// ---- POUs/CommonFB/MainFB/FB_CoupleAxis.TcPOU
(****************************************************************
NAME:			FB_CoupleAxis
DATA:			2017.2.16
VERSION:		1.0.0
DESCRIPTION:	FB_CoupleAxis
HISTORY:
				2017.2.16		NEW

***************************************************************)
FUNCTION_BLOCK FB_CoupleAxis
VAR_INPUT
	Execute:BOOL;
	Reset:BOOL;
END_VAR
VAR_OUTPUT
	FbID:DINT:=1001;
	State:DINT;
	Busy:BOOL;
	InGear:BOOL;
	Error:BOOL;
	ErrorID:DINT;
END_VAR
VAR_IN_OUT
END_VAR
VAR
	Bottom_MC_GearIn: MC_GearIn;
	Top_MC_GearIn: MC_GearIn;
	fb_ton: TON;
END_VAR

IF Execute THEN
Busy:=TRUE;
InGear:=FALSE;
fb_ton(PT:=t#0.1s);
CASE State OF
	0:	(*Check*)
		IF LeftTopLin.NcToPlc.CoupleState=3 OR LeftBottomLin.NcToPlc.CoupleState=3 THEN	
			ErrorID:=1;
			State:=-100;
		ELSIF LeftTopLin.NcToPlc.CoupleState=2 OR LeftBottomLin.NcToPlc.CoupleState=2
			OR RightTopLin.NcToPlc.CoupleState=2 OR RightBottomLin.NcToPlc.CoupleState=2 THEN
			ErrorID:=2;
			State:=-100;
		ELSIF LeftTopLin.NcToPlc.CoupleState=1 AND LeftBottomLin.NcToPlc.CoupleState=1
			AND RightTopLin.NcToPlc.CoupleState=3 AND RightBottomLin.NcToPlc.CoupleState=3 THEN	
			ErrorID:=3;
			State:=-100;
		ELSIF LeftTopLin.Status.Moving OR  RightTopLin.Status.Moving OR LeftBottomLin.Status.Moving OR RightBottomLin.Status.Moving THEN	(*ÓÐÖáÔË¶¯*)
			ErrorID:=4;
			State:=-100;
		ELSIF  Top_MC_GearIn.Error OR Bottom_MC_GearIn.Error THEN		(*FB Error*)
			ErrorID:=5;
			State:=99;
		ELSIF Top_MC_GearIn.InGear OR Bottom_MC_GearIn.InGear THEN
			ErrorID:=6;
			State:=99;
		ELSIF LeftTopLin.NcToPlc.CoupleState=0 AND LeftBottomLin.NcToPlc.CoupleState=0
			AND RightTopLin.NcToPlc.CoupleState=0 AND RightBottomLin.NcToPlc.CoupleState=0 THEN
			State:=1;
		ELSE
			ErrorID:=7;
			State:=-100;
		END_IF
	1:	(*Couple*)
		IF LeftTopLin.NcToPlc.CoupleState=0 AND LeftBottomLin.NcToPlc.CoupleState=0
			AND RightTopLin.NcToPlc.CoupleState=0 AND RightBottomLin.NcToPlc.CoupleState=0 THEN	
			Top_MC_GearIn.Execute:=TRUE;
			Bottom_MC_GearIn.Execute:=TRUE;
			A_CoupleMC();
			fb_ton.IN:=TRUE;
			State:=2;
		ELSE
			ErrorID:=7;
			State:=99;
		END_IF
	2:	(*Couple Wait*)
		A_CoupleMC();
		IF NOT Top_MC_GearIn.InGear OR NOT Bottom_MC_GearIn.InGear THEN	
			IF NOT fb_ton.Q THEN
				State:=2;
			ELSE
				ErrorID:=8;
				State:=99;
			END_IF
		ELSIF  LeftTopLin.NcToPlc.CoupleState<>1 OR  RightTopLin.NcToPlc.CoupleState<>3
			OR LeftBottomLin.NcToPlc.CoupleState<>1 OR  RightBottomLin.NcToPlc.CoupleState<>3 THEN	
				ErrorID:=9;
				State:=-100;
		ELSIF   LeftTopLin.NcToPlc.CoupleState=1 AND  RightTopLin.NcToPlc.CoupleState=3
			AND LeftBottomLin.NcToPlc.CoupleState=1 AND  RightBottomLin.NcToPlc.CoupleState=3 THEN	
				State:=88;
		ELSE
				ErrorID:=10;
				State:=-100;
		END_IF
	88:	(*InGear*)
		Execute:=FALSE;
		State:=0;
		Busy:=FALSE;
		InGear:=TRUE;
		Error:=FALSE;
		ErrorID:=0;
		Bottom_MC_GearIn.Execute:=FALSE;
		Top_MC_GearIn.Execute:=FALSE;
		A_CoupleMC();
		fb_ton.IN:=FALSE;
	99:	(*FB Error*)
		Execute:=FALSE;
		State:=99;
		Busy:=FALSE;
		InGear:=FALSE;
		Error:=TRUE;
		Bottom_MC_GearIn.Execute:=FALSE;
		Top_MC_GearIn.Execute:=FALSE;
		A_CoupleMC();
		fb_ton.IN:=FALSE;
	-100:	(*Emergency Error*)
		FB_PlcEmergencyStop();
		Execute:=FALSE;
		State:=-100;
		Busy:=FALSE;
		InGear:=FALSE;
		Error:=TRUE;
		Bottom_MC_GearIn.Execute:=FALSE;
		Top_MC_GearIn.Execute:=FALSE;
		A_CoupleMC();
		fb_ton.IN:=FALSE;
END_CASE
END_IF
IF Reset THEN
		Execute:=FALSE;
		State:=0;
		Busy:=FALSE;
		InGear:=FALSE;
		Error:=FALSE;
		ErrorID:=0;
		Bottom_MC_GearIn.Execute:=FALSE;
		Top_MC_GearIn.Execute:=FALSE;
		A_CoupleMC();
		Reset:=FALSE;
END_IF

ACTION A_CoupleMC:
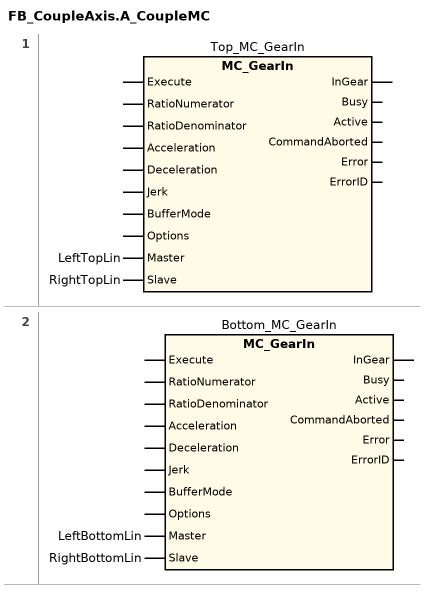
// NETWORK 1
Top_MC_GearIn(Master := LeftTopLin, Slave := RightTopLin); // MC_GearIn

// NETWORK 2
Bottom_MC_GearIn(Master := LeftBottomLin, Slave := RightBottomLin); // MC_GearIn
END_ACTION

END_FUNCTION_BLOCK

// ---- POUs/CommonFB/MainFB/FB_SetMotorAxisPosition.TcPOU
(****************************************************************
NAME:			FB_SetAxisPosition
DATA:			2017.2.16
VERSION:		1.0.0
DESCRIPTION:	FB_SetAxisPosition
HISTORY:
				2017.2.16		NEW

***************************************************************)
FUNCTION_BLOCK FB_SetMotorAxisPosition
VAR_INPUT
	//GapValueSet:LREAL:=0;
	ValueSet_LeftTop:LREAL:=0;
	ValueSet_RightTop:LREAL:=0;
	ValueSet_LeftBottom:LREAL:=0;
	ValueSet_RightBottom:LREAL:=0;
	Execute:BOOL;
END_VAR
VAR_OUTPUT
	FbID:DINT:=1001;
	State:DINT;
	Busy:BOOL;
	Done:BOOL;
	Error:BOOL;
	ErrorID:DINT;
END_VAR
VAR
	LeftTopMotor_MC_SetPosition: MC_SetPosition;
	RightTopMotor_MC_SetPosition: MC_SetPosition;
	LeftBottomMotor_MC_SetPosition: MC_SetPosition;
	RightBottomMotor_MC_SetPosition: MC_SetPosition;
	fb_ton: TON;
	FB_Couple_Axis: FB_CoupleAxis;
	FB_PlcEmergencyStop: FB_PlcEmergencyStop;
END_VAR

IF Execute THEN
Busy:=TRUE;
Done:=FALSE;
fb_ton(PT:=t#0.1s);
CASE State OF
	0:
		IF LeftTopMotor_MC_SetPosition.Error OR RightTopMotor_MC_SetPosition.Error
			OR LeftBottomMotor_MC_SetPosition.Error OR RightBottomMotor_MC_SetPosition.Error THEN		(*FB Error*)
			ErrorID:=1;
			State:=99;
		ELSIF FB_Couple_Axis.InGear THEN		
			ErrorID:=2;
			State:=99;
		ELSIF LeftTopMotor.NcToPlc.CoupleState=0 AND LeftBottomMotor.NcToPlc.CoupleState=0
			AND RightTopMotor.NcToPlc.CoupleState=0 AND RightBottomMotor.NcToPlc.CoupleState=0 THEN	
			State:=1;
		ELSE
			ErrorID:=3;
			State:=-100;
		END_IF
	1:	(*Execute*)
		LeftTopMotor_MC_SetPosition.Position:=ValueSet_LeftTop;
		LeftTopMotor_MC_SetPosition.Execute:=TRUE;
		RightTopMotor_MC_SetPosition.Position:=ValueSet_RightTop;
		RightTopMotor_MC_SetPosition.Execute:=TRUE;
		LeftBottomMotor_MC_SetPosition.Position:=ValueSet_LeftBottom;
		LeftBottomMotor_MC_SetPosition.Execute:=TRUE;
		RightBottomMotor_MC_SetPosition.Position:=ValueSet_RightBottom;
		RightBottomMotor_MC_SetPosition.Execute:=TRUE;
		A_SetMotorPositionMC();
		fb_ton.IN:=TRUE;
		State:=2;
	2:	(*Wait*)
		A_SetMotorPositionMC();
		IF NOT LeftTopMotor_MC_SetPosition.Done OR NOT RightTopMotor_MC_SetPosition.Done
			OR NOT LeftBottomMotor_MC_SetPosition.Done OR NOT RightBottomMotor_MC_SetPosition.Done THEN		
			IF NOT fb_ton.Q THEN
				State:=2;
			ELSE
				ErrorID:=4;
				State:=99;
			END_IF
		ELSIF  LeftTopMotor_MC_SetPosition.Done AND RightTopMotor_MC_SetPosition.Done
			AND LeftBottomMotor_MC_SetPosition.Done AND RightBottomMotor_MC_SetPosition.Done THEN		
			State:=88;
		ELSE
			ErrorID:=5;
			State:=99;
		END_IF
	88:
		Execute:=FALSE;
		State:=0;
		Busy:=FALSE;
		Done:=TRUE;
		Error:=FALSE;
		ErrorID:=0;
		LeftTopMotor_MC_SetPosition.Execute:=FALSE;
		RightTopMotor_MC_SetPosition.Execute:=FALSE;
		LeftBottomMotor_MC_SetPosition.Execute:=FALSE;
		RightBottomMotor_MC_SetPosition.Execute:=FALSE;
		fb_ton.IN:=FALSE;
	99:
		Execute:=FALSE;
		State:=99;
		Busy:=FALSE;
		Done:=FALSE;
		Error:=TRUE;
		LeftTopMotor_MC_SetPosition.Execute:=FALSE;
		RightTopMotor_MC_SetPosition.Execute:=FALSE;
		LeftBottomMotor_MC_SetPosition.Execute:=FALSE;
		RightBottomMotor_MC_SetPosition.Execute:=FALSE;
		fb_ton.IN:=FALSE;
	-100:
		FB_PlcEmergencyStop();
		Execute:=FALSE;
		State:=-100;
		Busy:=FALSE;
		Done:=FALSE;
		Error:=TRUE;
		LeftTopMotor_MC_SetPosition.Execute:=FALSE;
		RightTopMotor_MC_SetPosition.Execute:=FALSE;
		LeftBottomMotor_MC_SetPosition.Execute:=FALSE;
		RightBottomMotor_MC_SetPosition.Execute:=FALSE;
		fb_ton.IN:=FALSE;
END_CASE
END_IF

ACTION A_SetMotorPositionMC:
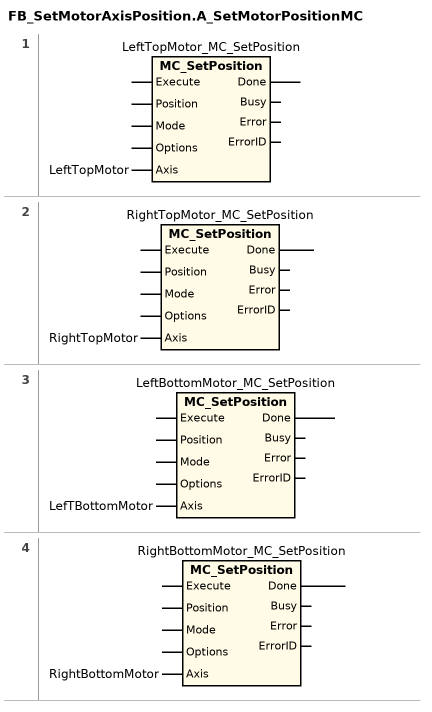
// NETWORK 1
LeftTopMotor_MC_SetPosition(Axis := LeftTopMotor); // MC_SetPosition

// NETWORK 2
RightTopMotor_MC_SetPosition(Axis := RightTopMotor); // MC_SetPosition

// NETWORK 3
LeftBottomMotor_MC_SetPosition(Axis := LefTBottomMotor); // MC_SetPosition

// NETWORK 4
RightBottomMotor_MC_SetPosition(Axis := RightBottomMotor); // MC_SetPosition
END_ACTION

END_FUNCTION_BLOCK

// ---- POUs/1.CarrierMode/SingleCarrierMode/SingleCarrierMode.TcPOU
PROGRAM SingleCarrierMode
VAR
	TopPositionNew:LREAL:=100;
	TopVelocityNew:LREAL:=0.02;
	btn_TopMove:BOOL;
	btn_TopStop:BOOL;
	BottomPositionNew:LREAL:=100;
	BottomVelocityNew:LREAL:=0.02;
	btn_BottomMove:BOOL;
	btn_BottomStop:BOOL;
	(*Var*)
	fb_ton1:TON;
	fb_ton2:TON;
	fb_ton3:TON;
	(*Status*)
	State:DINT;
	Busy:BOOL;
	TopBusy:BOOL;
	BottomBusy:BOOL;
	InitDone:BOOL;
	tm_state: DINT;
	ts_state: DINT;
	bm_state: DINT;
	bs_state: DINT;
	moni_State:DINT;
	(*PowerOff*)
	d_state: DINT;
	(*¼ì²âµ½ÏÞÎ»£¬»Ö¸´Move×´Ì¬*)
	FTrig_ReachLS: F_TRIG;
	FTrig_btn_GapMove: F_TRIG;
	InitPowerDone:BOOL;
END_VAR

TopPositionActual:=(Pos_LeftTopLin+Pos_RightTopLin)/2;
TopVelocityActual:=(Velo_LeftTopLin+Velo_RightTopLin)/2;
BottomPositionActual:=(Pos_LeftBottomLin+Pos_RightBOttomLin)/2;
BottomVelocityActual:=(Velo_LeftBottomLin+Velo_RightBOttomLin)/2;
(*btn_Power On/Off*)
IF btn_Power AND st_Power=0 THEN
	btn_PowerOn:=TRUE;
	btn_Power:=FALSE;
END_IF
IF btn_Power AND st_Power=1 THEN
	btn_PowerOff:=TRUE;
	btn_Power:=FALSE;
END_IF
IF btn_PowerOn THEN
	A_PowerOn();
END_IF
IF btn_PowerOff THEN
	A_PowerOff();
END_IF

(*********************************************************************Monitor All Carrirt Position***********************************************)
A_MonitoringAllAxis();
(*********************************************************************btn_TopMove*****************************************************************)
IF btn_TopMove AND NOT bottomBusy THEN
		TopBusy:=TRUE;
		btn_BottomMove:=FALSE;
		IF NOT st_Power THEN
			ErrorID:=1501;
			Error:=TRUE;
			ErrorDescription:='Plz PowerOn Frist';
			LED_Error:=TRUE;
			RETURN;
		ELSE
			ErrorID:=0;
			Error:=FALSE;
			ErrorDescription:='';
			LED_Error:=FALSE;
		END_IF
		CASE tm_state OF
			0:
				FB_Move.Mode:=2;						(*单梁模式*)
				FB_Move.CoupleState:=st_Couple;			
				FB_Move.PowerState:=st_Power;			
				FB_Move.TopMove:=TRUE;				
				FB_Move.TopPosition:=TopPositionNew;		
				FB_Move.TopVelocity:=TopVelocityNew;		
				FB_Move();								
				tm_state:=1;
			1:
				FB_Move();
				LED_Run:=TRUE;
				IF NOT FB_Move.TopDone THEN	
					tm_state:=1;
				ELSE					
					tm_state:=88;
				END_IF
			88:
				btn_TopMove:=FALSE;	
				LED_Run:=FALSE;
				tm_state:=0;
				TopBusy:=FALSE;
		END_CASE
END_IF

(*********************************************************************btn_BottomMove*****************************************************************)
IF btn_BottomMove AND NOT TopBusy THEN
		btn_TopMove:=FALSE;
		BottomBusy:=TRUE;
		IF NOT st_Power THEN
			ErrorID:=1501;
			Error:=TRUE;
			ErrorDescription:='Plz PowerOn Frist';
			LED_Error:=TRUE;
			RETURN;
		ELSE
			ErrorID:=0;
			Error:=FALSE;
			ErrorDescription:='';
			LED_Error:=FALSE;
		END_IF
		CASE bm_state OF
			0:
				FB_Move.Mode:=2;						
				FB_Move.CoupleState:=st_Couple;			
				FB_Move.PowerState:=st_Power;			
				FB_Move.BottomMove:=TRUE;			
				FB_Move.BottomPosition:=BottomPositionNew;		
				FB_Move.BottomVelocity:=BottomVelocityNew;		
				FB_Move();
				bm_state:=1;
			1:
				FB_Move();
				IF NOT FB_Move.BottomDone THEN
					LED_Run:=TRUE;
					bm_state:=1;
				ELSE
					bm_state:=88;
				END_IF
			88:
				BottomBusy:=FALSE;
				btn_TopMove:=FALSE;
				btn_BottomMove:=FALSE;
				bm_state:=0;
				LED_Run:=FALSE;
		END_CASE
END_IF
(*******************************************************************btn_TopStop********************************************************************)

IF btn_TopStop OR btn_reset THEN
	LED_Run:=FALSE;
	TopMoveIndicator:=0;
	FB_Move.TopReset:=TRUE;
	TopBusy:=FALSE;
	FB_Move();
	btn_TopMove:=FALSE;	
	tm_state:=0;
	CASE ts_state OF
			0:
				FB_Stop.Mode:=2;
				FB_Stop.CoupleState:=st_Couple;
				FB_Stop.PowerState:=st_Power;
				FB_Stop.TopStop:=TRUE;	
				FB_Stop();	
				ts_state:=1;
			1:
				FB_Stop();
				IF NOT FB_Stop.TopDone THEN
					ts_state:=1;
				ELSE
					ts_state:=88;
				END_IF
			88:
				btn_TopStop:=FALSE;	
				FB_Move.TopReset:=FALSE;	
				ts_state:=0;
				btn_reset:=FALSE;
		END_CASE
END_IF
(*******************************************************************btn_BottomStop********************************************************************)
IF btn_BottomStop OR btn_reset THEN
	LED_Run:=FALSE;
	BottomMoveIndicator:=0;
	FB_Move.BottomReset:=TRUE;
	BottomBusy:=FALSE;
	FB_Move();			
	btn_BottomMove:=FALSE;			
	bm_state:=0;							
	CASE bs_state OF
			0:
				FB_Stop.Mode:=2;							
				FB_Stop.CoupleState:=st_Couple;			
				FB_Stop.PowerState:=st_Power;			
				FB_Stop.BottomStop:=TRUE;				
				FB_Stop();								
				bs_state:=1;
			1:
				FB_Stop();
				IF NOT FB_Stop.BottomDone THEN		
					bs_state:=1;
				ELSE									
					bs_state:=88;
				END_IF
			88:
				btn_BottomStop:=FALSE;					
				FB_Move.BottomReset:=FALSE;				
				bs_state:=0;
				btn_reset:=FALSE;
		END_CASE
END_IF
(************************************************************************************************************************)

FTrig_ReachLS(CLK:=Unreach_LS_Far AND Unreach_LS_Near);
IF FTrig_ReachLS.Q THEN		
	btn_TopStop:=TRUE;
	btn_BottomStop:=TRUE;
END_IF
IF btn_TopStop THEN			
	btn_BottomStop:=TRUE;
END_IF

ACTION A_MonitoringAllAxis:
(****************************************************************
NAME:			A_MonitoringAllAxis
DATA:			2017.3.20
VERSION:		1.0.0
DESCRIPTION:	

HISTORY:
				2017.3.20		NEW

***************************************************************)
IF  st_Power<>0 THEN
		Diff_TopPos_actual:=Pos_leftTopLin-Pos_RightTopLin;
		Diff_TopVelo_actual:=Velo_leftTopLin-Velo_RightTopLin;
IF ABS(Pos_leftTopLin-Pos_RightTopLin)>Threshold_TopPos_SingleCarrier THEN
		btn_TopStop:=TRUE;
		btn_BottomStop:=TRUE;
		FB_PlcEmergencyStop();
		Error:=TRUE;
		ErrorID:=14;
		LED_Error:=TRUE;
ELSIF ABS(Velo_leftTopLin-Velo_RightTopLin)>Threshold_TopVelo_SingleCarrier  THEN
		(*btn_TopStop:=TRUE;
		btn_BottomStop:=TRUE;
		FB_PlcEmergencyStop();*)
		Error:=TRUE;
		ErrorID:=15;

ELSIF ABS(Pos_LeftBottomLin-Pos_RightBottomLin)>Threshold_BottomPos_SingleCarrier THEN
		btn_TopStop:=TRUE;
		btn_BottomStop:=TRUE;
		FB_PlcEmergencyStop();
		Error:=TRUE;
		ErrorID:=16;
		LED_Error:=TRUE;
ELSIF ABS(Velo_leftBottomLin-Velo_RightBottomLin)>Threshold_BottomVelo_SingleCarrier  THEN
		(*btn_TopStop:=TRUE;
		btn_BottomStop:=TRUE;
		FB_PlcEmergencyStop();*)
		Error:=TRUE;
		ErrorID:=17;

END_IF
END_IF
(**************************************************************************************************************************************)
END_ACTION

ACTION A_PowerOff:
CASE d_state OF
		0:(*PowerOff*)
			FB_Power(Off:=TRUE);
				d_state:=1;
		1:
			IF NOT FB_power.OffStatus THEN
				d_state:=1;
			ELSE
				d_state:=88;
			END_IF
		88:(*ResetAllState*)
			btn_PowerOn:=FALSE;
			btn_TopMove:=FALSE;
			btn_TopStop:=FALSE;
			btn_BottomMove:=FALSE;
			btn_BottomStop:=FALSE;
			LeftTopLinMoveIndicator:=0;
			RightTopLinMoveIndicator:=0;
			LeftBottomLinMoveIndicator:=0;
			RightBottomLinMoveIndicator:=0;
			fb_ton1.IN:=FALSE;
			fb_ton2.IN:=FALSE;
			fb_ton3.IN:=FALSE;
			State:=0;
			Busy:=FALSE;
			InitPowerDone:=FALSE;
			Error:=FALSE;
			ErrorID:=0;
			tm_state:=0;
			ts_state:=0;
			bm_state:=0;
			bs_state:=0;
			btn_PowerOff:=FALSE;
			d_state:=0;
			Led_Run:=FALSE;
			Led_Error:=FALSE;
			moni_State:=0;
END_CASE
END_ACTION

ACTION A_PowerOn:
(****************************************************************
NAME:			A_PowerOn
DATA:			2018.1.9
VERSION:		1.0.0
DESCRIPTION:	

HISTORY:
				2019.1.9		NEW

***************************************************************)
fb_ton3(PT:=t#0.5s);
CASE State OF
	0:	(*FB_Power_On*)
		FB_Power(On:=TRUE);
		fb_ton3.IN:=TRUE;
		State:=1;
	1:	(*wait*)
		FB_power();
		IF NOT FB_power.OnStatus THEN
			IF NOT fb_ton3.Q THEN
				State:=1;
			ELSE
				ErrorID:=1;
				State:=99;
			END_IF
		ELSE
			State:=88;
		END_IF
	88:	(*All Done*)
		btn_PowerOn:=FALSE;
		State:=0;
		Error:=FALSE;
		ErrorID:=0;
		Busy:=FALSE;
		InitPowerDone:=TRUE;
		FB_power.On:=FALSE;
		fb_ton3.IN:=FALSE;
		LED_Error:=FALSE;
	99:
		Error:=TRUE;
		//ErrorID:=701;
		//ErrorDescription:='power on error';		
		btn_PowerOn:=FALSE;
		State:=99;
		Busy:=FALSE;
		InitPowerDone:=FALSE;
		fb_ton3.IN:=FALSE;
		LED_Error:=TRUE;
END_CASE
END_ACTION

END_PROGRAM

// ---- POUs/CommonFB/MainFB/FB_Move.TcPOU
(****************************************************************
NAME:			FB_Move
DATA:			2017.2.17
VERSION:		1.0.0
DESCRIPTION:	FB_Move
HISTORY:
				2017.2.17		NEW
				2018.1.9		ÐÂÔöBCGapMode
***************************************************************)
FUNCTION_BLOCK FB_Move
VAR_INPUT
	(*È«¾Ö*)
	Mode:DINT;
	PowerState:BOOL;
	CoupleState:DINT;
	(*BCGapMode*)
	BCLeftTopPosition:LREAL;
	BCLeftTopVelocity:LREAL;
	BCRightTopPosition:LREAL;
	BCRightTopVelocity:LREAL;
	BCLeftBottomPosition:LREAL;
	BCLeftBottomVelocity:LREAL;
	BCRightBottomPosition:LREAL;
	BCRightBottomVelocity:LREAL;
	BCGapMove:BOOL;
	BCGapReset:BOOL;
	BCGapMove_2:BOOL;
	BCGapReset_2:BOOL;
	(*GapMode*)
	GapPosition:LREAL;
	GapVelocity:LREAL;
	GapMove:BOOL;
	GapReset:BOOL;
	(*SingleCarrierMode*)
	TopPosition:LREAL;
	TopVelocity:LREAL;
	TopMove:BOOL;
	TopReset:BOOL;
	BottomPosition:LREAL;
	BottomVelocity:LREAL;
	BottomMove:BOOL;
	BottomReset:BOOL;
	(*TaperMode*)
	TaperPosition:LREAL;
	TaperVelocity:LREAL;
	TaperMove:BOOL;
	TaperStop:BOOL;
	TaperReset:BOOL;
	(**DebugMode*)
	LeftTopPosition:LREAL;
	LeftTopVelocity:LREAL;
	LeftTopMove:BOOL;
	LeftTopStop:BOOL;
	LeftTopReset:BOOL;
	RightTopPosition:LREAL;
	RightTopVelocity:LREAL;
	RightTopMove:BOOL;
	RightTopStop:BOOL;
	RightTopReset:BOOL;
	LeftBottomPosition:LREAL;
	LeftBottomVelocity:LREAL;
	LeftBottomMove:BOOL;
	LeftBottomStop:BOOL;
	LeftBottomReset:BOOL;
	RightBottomPosition:LREAL;
	RightBottomVelocity:LREAL;
	RightBottomMove:BOOL;
	RightBottomStop:BOOL;
	RightBottomReset:BOOL;
END_VAR
VAR_OUTPUT
	FbID:DINT:=1001;
	GapState:DINT;
	GapBusy:BOOL;
	GapDone:BOOL;
	GapMoving:BOOL;

	BCGapState:DINT;
	BCGapBusy:BOOL;
	BCGapDone:BOOL;

	TopState:DINT;
	TopBusy:BOOL;
	TopDone:BOOL;
	BottomState:DINT;
	BottomBusy:BOOL;
	BottomDone:BOOL;

	TaperState:DINT;
	TaperBusy:BOOL;
	TaperDone:BOOL;

	LeftTopState:DINT;
	LeftTopBusy:BOOL;
	LeftTopDone:BOOL;
	RightTopState:DINT;
	RightTopBusy:BOOL;
	RightTopDone:BOOL;
	LeftBottomState:DINT;
	LeftBottomBusy:BOOL;
	LeftBottomDone:BOOL;
	RightBottomState:DINT;
	RightBottomBusy:BOOL;
	RightBottomDone:BOOL;


	Error:BOOL;
	ErrorID:DINT;
	
	GapState_2:DINT;
	GapBusy_2:BOOL;
	GapDone_2:BOOL;

	BCGapState_2:DINT;
	BCGapBusy_2:BOOL;
	BCGapDone_2:BOOL;
END_VAR
VAR
	Top_MC_MoveAbsolute: MC_MoveAbsolute;
	Bottom_MC_MoveAbsolute: MC_MoveAbsolute;
	RightTopLin_MC_MoveAbsolute: MC_MoveAbsolute;
	RightBottomLin_MC_MoveAbsolute: MC_MoveAbsolute;
	fb_ton: TON;
	fb_ton1: TON;
	fb_ton2: TON;
	fb_ton_debug_1:TON;
	fb_ton_debug_2:TON;
	fb_ton_debug_3:TON;
	fb_ton_debug_4:TON;
	fb_ton_BC:TON;
	fb_ton_BC_2:TON;
END_VAR

IF PowerState=1 THEN
	IF Mode=1 AND CoupleState=1 THEN
		A_GapMove();
	ELSIF Mode=2 AND CoupleState=0 AND TopMove THEN
		A_TopMove();
	ELSIF Mode=2 AND CoupleState=0 AND BottomMove THEN
		A_BottomMove();
	ELSIF Mode=3 AND CoupleState=0 AND TaperMove THEN
		A_TaperMove();
	ELSIF Mode=4 AND CoupleState=0 AND LeftTopMove THEN
		A_LeftTopMove();
	ELSIF Mode=4 AND CoupleState=0 AND RightTopMove THEN
		A_RightTopMove();
	ELSIF Mode=4 AND CoupleState=0 AND LeftBottomMove THEN
		A_LeftBottomMove();
	ELSIF Mode=4 AND CoupleState=0 AND RightBottomMove THEN
		A_RightBottomMove();
	ELSIF Mode=5 AND CoupleState=0 AND BCGapMove THEN
		A_BCGapMove();
	ELSIF Mode=6 AND CoupleState=0 AND BCGapMove_2 THEN
		A_BCGapMove_2();
	END_IF
END_IF

ACTION A_BCGapMove:
IF BCGapMove THEN
BCGapBusy:=TRUE;
BCGapDone:=FALSE;
fb_ton_BC(PT:=T#80S);(*2mm/s max spees,120mm*)

IF LeftTopLin.NcToPlc.CoupleState<>0 OR LeftBottomLin.NcToPlc.CoupleState<>0
			OR RightTopLin.NcToPlc.CoupleState<>0 OR RightBottomLin.NcToPlc.CoupleState<>0 THEN
			ErrorID:=1;
			GapState:=-100;
END_IF
A_MoveMC();
IF  LeftTopLin.Status.Moving AND RightTopLin.Status.Moving
			 AND LeftBottomLin.Status.Moving AND RightBottomLin.Status.Moving THEN
	GapMoving:=TRUE;
ELSE
	GapMoving:=FALSE;
END_IF
CASE BCGapState OF
	0:
		IF LeftTopLin.Status.Moving OR RightTopLin.Status.Moving
			 OR LeftBottomLin.Status.Moving OR RightBottomLin.Status.Moving THEN	
			BCGapState:=88;
		//ELSIF Top_MC_MoveAbsolute.Error OR Bottom_MC_MoveAbsolute.Error OR
		//		RightTopLin_MC_MoveAbsolute.Error OR RightBottomLin_MC_MoveAbsolute.Error THEN	
		//	ErrorID:=2;
		//	BCGapState:=99;
		(*ELSIF ABS(Pos_LeftTopLin-GapPosition/2)<0.002 AND  ABS(Pos_LeftBottomLin-GapPosition)<0.002 THEN	
			GapState:=88;*)
		ELSIF leftTopLin.Status.NotMoving AND  leftBottomLin.Status.NotMoving
			 AND RightTopLin.Status.NotMoving AND RightBottomLin.Status.NotMoving THEN	
			BCGapState:=1;
		END_IF
	1:
		Top_MC_MoveAbsolute.Position:=BCLeftTopPosition;
		Top_MC_MoveAbsolute.Velocity:=BCLeftTopVelocity;
		Bottom_MC_MoveAbsolute.Position:=BCLeftBottomPosition;
		Bottom_MC_MoveAbsolute.Velocity:=BCLeftBottomVelocity;
		RightTopLin_MC_MoveAbsolute.Position:=BCRightTopPosition;
		RightTopLin_MC_MoveAbsolute.Velocity:=BCRightTopVelocity;
		RightBottomLin_MC_MoveAbsolute.Position:=BCRightBottomPosition;
		RightBottomLin_MC_MoveAbsolute.Velocity:=BCRightBottomVelocity;
		Top_MC_MoveAbsolute.Execute:=TRUE;
		Bottom_MC_MoveAbsolute.Execute:=TRUE;
		RightTopLin_MC_MoveAbsolute.Execute:=TRUE;
		RightBottomLin_MC_MoveAbsolute.Execute:=TRUE;
		fb_ton_BC.IN:=TRUE;
		BCGapState:=2;
	2:
		IF NOT Top_MC_MoveAbsolute.Done OR NOT  Bottom_MC_MoveAbsolute.Done
				OR NOT RightTopLin_MC_MoveAbsolute.Done OR NOT RightBottomLin_MC_MoveAbsolute.Done THEN	
			BCGapState:=2;
		ELSIF Top_MC_MoveAbsolute.Done  AND  Bottom_MC_MoveAbsolute.Done AND RightTopLin_MC_MoveAbsolute.Done AND RightBottomLin_MC_MoveAbsolute.Done THEN		(*ÔË¶¯Íê³É£¬×ªÏÂÒ»²½*)
			BCGapState:=88;
		END_IF
		(*½ÓÊÕµ½stopÐÅºÅÊ±£¬reset×´Ì¬*)
		IF BCGapReset THEN
			BCGapState:=88;
		END_IF

	88:
		BCGapMove:=FALSE;
		BCGapState:=0;
		BCGapBusy:=FALSE;
		BCGapDone:=TRUE;
		Error:=FALSE;
		ErrorID:=0;
		Top_MC_MoveAbsolute.Execute:=FALSE;
		Bottom_MC_MoveAbsolute.Execute:=FALSE;
		RightTopLin_MC_MoveAbsolute.Execute:=FALSE;
		RightBottomLin_MC_MoveAbsolute.Execute:=FALSE;
		fb_ton_BC.IN:=FALSE;
	89:
		BCGapMove:=FALSE;
		BCGapState:=0;
		BCGapBusy:=FALSE;
		BCGapDone:=FALSE;
		Error:=FALSE;
		ErrorID:=0;
		Top_MC_MoveAbsolute.Execute:=FALSE;
		Bottom_MC_MoveAbsolute.Execute:=FALSE;
		RightTopLin_MC_MoveAbsolute.Execute:=FALSE;
		RightBottomLin_MC_MoveAbsolute.Execute:=FALSE;
		fb_ton_BC.IN:=FALSE;
	99:
		BCGapMove:=FALSE;
		BCGapState:=0;
		BCGapBusy:=FALSE;
		BCGapDone:=FALSE;
		Error:=TRUE;
		Top_MC_MoveAbsolute.Execute:=FALSE;
		Bottom_MC_MoveAbsolute.Execute:=FALSE;
		RightTopLin_MC_MoveAbsolute.Execute:=FALSE;
		RightBottomLin_MC_MoveAbsolute.Execute:=FALSE;
		fb_ton_BC.IN:=FALSE;
	-100:
		FB_PlcEmergencyStop();
		BCGapMove:=FALSE;
		BCGapState:=-100;
		BCGapBusy:=FALSE;
		BCGapDone:=FALSE;
		Error:=TRUE;
		Top_MC_MoveAbsolute.Execute:=FALSE;
		Bottom_MC_MoveAbsolute.Execute:=FALSE;
		RightTopLin_MC_MoveAbsolute.Execute:=FALSE;
		RightBottomLin_MC_MoveAbsolute.Execute:=FALSE;
		fb_ton_BC.IN:=FALSE;
END_CASE
END_IF
END_ACTION

ACTION A_BCGapMove_2:
IF BCGapMove_2 THEN
BCGapBusy_2:=TRUE;
BCGapDone_2:=FALSE;
fb_ton_BC_2(PT:=T#80S);(*2mm/s max spees,120mm*)
IF LeftTopLin.NcToPlc.CoupleState<>0 OR LeftBottomLin.NcToPlc.CoupleState<>0
			OR RightTopLin.NcToPlc.CoupleState<>0 OR RightBottomLin.NcToPlc.CoupleState<>0 THEN
			ErrorID:=1;
			GapState:=-100;
END_IF
A_MoveMC();
CASE BCGapState_2 OF
	0:
		IF LeftTopLin.Status.Moving OR RightTopLin.Status.Moving
			 OR LeftBottomLin.Status.Moving OR RightBottomLin.Status.Moving THEN	
			BCGapState_2:=88;
		ELSIF Top_MC_MoveAbsolute.Error OR Bottom_MC_MoveAbsolute.Error OR
				RightTopLin_MC_MoveAbsolute.Error OR RightBottomLin_MC_MoveAbsolute.Error THEN	
			ErrorID:=2;
			BCGapState_2:=99;
		(*ELSIF ABS(Pos_LeftTopLin-GapPosition/2)<0.002 AND  ABS(Pos_LeftBottomLin-GapPosition)<0.002 THEN	
			GapState:=88;*)
		ELSIF leftTopLin.Status.NotMoving AND  leftBottomLin.Status.NotMoving
			 AND RightTopLin.Status.NotMoving AND RightBottomLin.Status.NotMoving THEN
			BCGapState_2:=1;
		END_IF
	1:
		Top_MC_MoveAbsolute.Position:=BCLeftTopPosition;
		Top_MC_MoveAbsolute.Velocity:=BCLeftTopVelocity;
		Bottom_MC_MoveAbsolute.Position:=BCLeftBottomPosition;
		Bottom_MC_MoveAbsolute.Velocity:=BCLeftBottomVelocity;
		RightTopLin_MC_MoveAbsolute.Position:=BCRightTopPosition;
		RightTopLin_MC_MoveAbsolute.Velocity:=BCRightTopVelocity;
		RightBottomLin_MC_MoveAbsolute.Position:=BCRightBottomPosition;
		RightBottomLin_MC_MoveAbsolute.Velocity:=BCRightBottomVelocity;
		Top_MC_MoveAbsolute.Execute:=TRUE;
		Bottom_MC_MoveAbsolute.Execute:=TRUE;
		RightTopLin_MC_MoveAbsolute.Execute:=TRUE;
		RightBottomLin_MC_MoveAbsolute.Execute:=TRUE;
		fb_ton_BC_2.IN:=TRUE;
		BCGapState_2:=2;
	2:
		IF NOT Top_MC_MoveAbsolute.Done OR NOT  Bottom_MC_MoveAbsolute.Done
				OR NOT RightTopLin_MC_MoveAbsolute.Done OR NOT RightBottomLin_MC_MoveAbsolute.Done THEN		
			BCGapState_2:=2;
		ELSIF Top_MC_MoveAbsolute.Done  AND  Bottom_MC_MoveAbsolute.Done AND RightTopLin_MC_MoveAbsolute.Done AND RightBottomLin_MC_MoveAbsolute.Done THEN		(*ÔË¶¯Íê³É£¬×ªÏÂÒ»²½*)
			BCGapState_2:=88;
		END_IF
		(*½ÓÊÕµ½stopÐÅºÅÊ±£¬reset×´Ì¬*)
		IF BCGapReset_2 THEN
			BCGapState_2:=89;
		END_IF

	88:
		BCGapMove_2:=FALSE;
		BCGapState_2:=0;
		BCGapBusy_2:=FALSE;
		BCGapDone_2:=TRUE;
		Error:=FALSE;
		ErrorID:=0;
		Top_MC_MoveAbsolute.Execute:=FALSE;
		Bottom_MC_MoveAbsolute.Execute:=FALSE;
		RightTopLin_MC_MoveAbsolute.Execute:=FALSE;
		RightBottomLin_MC_MoveAbsolute.Execute:=FALSE;
		fb_ton_BC_2.IN:=FALSE;
	89:
		BCGapMove_2:=FALSE;
		BCGapState_2:=0;
		BCGapBusy_2:=FALSE;
		BCGapDone_2:=FALSE;
		Error:=FALSE;
		ErrorID:=0;
		Top_MC_MoveAbsolute.Execute:=FALSE;
		Bottom_MC_MoveAbsolute.Execute:=FALSE;
		RightTopLin_MC_MoveAbsolute.Execute:=FALSE;
		RightBottomLin_MC_MoveAbsolute.Execute:=FALSE;
		fb_ton_BC_2.IN:=FALSE;
	99:
		BCGapMove_2:=FALSE;
		BCGapState_2:=99;
		BCGapBusy_2:=FALSE;
		BCGapDone_2:=FALSE;
		Error:=TRUE;
		Top_MC_MoveAbsolute.Execute:=FALSE;
		Bottom_MC_MoveAbsolute.Execute:=FALSE;
		RightTopLin_MC_MoveAbsolute.Execute:=FALSE;
		RightBottomLin_MC_MoveAbsolute.Execute:=FALSE;
		fb_ton_BC_2.IN:=FALSE;
	-100:
		FB_PlcEmergencyStop();
		BCGapMove_2:=FALSE;
		BCGapState_2:=-100;
		BCGapBusy_2:=FALSE;
		BCGapDone_2:=FALSE;
		Error:=TRUE;
		Top_MC_MoveAbsolute.Execute:=FALSE;
		Bottom_MC_MoveAbsolute.Execute:=FALSE;
		RightTopLin_MC_MoveAbsolute.Execute:=FALSE;
		RightBottomLin_MC_MoveAbsolute.Execute:=FALSE;
		fb_ton_BC_2.IN:=FALSE;
END_CASE
END_IF
END_ACTION

ACTION A_BottomMove:
IF BottomMove THEN
BottomBusy:=TRUE;
BottomDone:=FALSE;
fb_ton2(PT:=T#80S);(*2mm/s max spees,120mm*)
A_MoveMC();
CASE BottomState OF

	0:
		IF LeftTopLin.Status.Moving OR RightTopLin.Status.Moving
			 OR LeftBottomLin.Status.Moving OR RightBottomLin.Status.Moving THEN	
			TopState:=88;
		ELSIF  Bottom_MC_MoveAbsolute.Error OR RightBottomLin_MC_MoveAbsolute.Error THEN		
			ErrorID:=2;
			BottomState:=99;
		ELSIF leftTopLin.Status.NotMoving AND  leftBottomLin.Status.NotMoving
			 AND RightTopLin.Status.NotMoving AND RightBottomLin.Status.NotMoving THEN	
			BottomState:=1;
		END_IF
	1:
		Bottom_MC_MoveAbsolute.Position:=BottomPosition;
		Bottom_MC_MoveAbsolute.Velocity:=BottomVelocity;
		Bottom_MC_MoveAbsolute.Execute:=TRUE;
		RightBottomLin_MC_MoveAbsolute.Position:=BottomPosition;
		RightBottomLin_MC_MoveAbsolute.Velocity:=BottomVelocity;
		RightBottomLin_MC_MoveAbsolute.Execute:=TRUE;
		fb_ton2.IN:=TRUE;
		BottomState:=2;
	2:
		IF leftTopLin.Status.Moving OR RightTopLin.Status.Moving THEN	
			ErrorID:=3;
			BottomState:=-100;
		ELSIF  (LeftBottomLin.Status.Moving AND  RightBottomLin.Status.NotMoving)
				OR (RightBottomLin.Status.Moving AND  LeftBottomLin.Status.NotMoving) THEN
			//ErrorID:=4;
			//BottomState:=-100;
		ELSIF NOT Bottom_MC_MoveAbsolute.Done THEN		
			BottomState:=2;
		ELSIF Bottom_MC_MoveAbsolute.Done THEN		
				BottomState:=88;
		END_IF
		(*½ÓÊÕµ½stopÐÅºÅÊ±£¬reset×´Ì¬*)
		IF BottomReset THEN
			BottomState:=89;
		END_IF

	88:
		BottomMove:=FALSE;
		BottomState:=0;
		BottomBusy:=FALSE;
		BottomDone:=TRUE;
		Error:=FALSE;
		ErrorID:=0;
		Bottom_MC_MoveAbsolute.Execute:=FALSE;
		RightBottomLin_MC_MoveAbsolute.Execute:=FALSE;
		fb_ton2.IN:=FALSE;
	89:
		BottomMove:=FALSE;
		BottomState:=0;
		BottomBusy:=FALSE;
		BottomDone:=FALSE;
		Error:=FALSE;
		ErrorID:=0;
		Bottom_MC_MoveAbsolute.Execute:=FALSE;
		RightBottomLin_MC_MoveAbsolute.Execute:=FALSE;
		fb_ton2.IN:=FALSE;
	99:
		BottomMove:=FALSE;
		BottomState:=99;
		BottomBusy:=FALSE;
		BottomDone:=FALSE;
		Error:=TRUE;
		Bottom_MC_MoveAbsolute.Execute:=FALSE;
		RightBottomLin_MC_MoveAbsolute.Execute:=FALSE;
		fb_ton2.IN:=FALSE;
	-100:
		FB_PlcEmergencyStop();
		BottomMove:=FALSE;
		BottomState:=-100;
		BottomBusy:=FALSE;
		BottomDone:=FALSE;
		Error:=TRUE;
		Bottom_MC_MoveAbsolute.Execute:=FALSE;
		RightBottomLin_MC_MoveAbsolute.Execute:=FALSE;
		fb_ton2.IN:=FALSE;
END_CASE
END_IF
END_ACTION

ACTION A_GapMove:
IF GapMove THEN
GapBusy:=TRUE;
GapDone:=FALSE;
fb_ton(PT:=T#80S);(*2mm/s max spees,120mm*)

IF LeftTopLin.NcToPlc.CoupleState<>1 OR LeftBottomLin.NcToPlc.CoupleState<>1
			OR RightTopLin.NcToPlc.CoupleState<>3 OR RightBottomLin.NcToPlc.CoupleState<>3 THEN
			ErrorID:=1;
			GapState:=-100;
END_IF
A_MoveMC();
CASE GapState OF

	0:
		IF LeftTopLin.Status.Moving OR RightTopLin.Status.Moving
			 OR LeftBottomLin.Status.Moving OR RightBottomLin.Status.Moving THEN	
			GapState:=88;
		ELSIF Top_MC_MoveAbsolute.Error OR Bottom_MC_MoveAbsolute.Error THEN		
			ErrorID:=2;
			GapState:=99;
		ELSIF ABS(Pos_LeftTopLin-GapPosition/2)<0.002 AND  ABS(Pos_LeftBottomLin-GapPosition)<0.002 THEN	
			GapState:=88;
		ELSIF leftTopLin.Status.NotMoving AND  leftBottomLin.Status.NotMoving
			 AND RightTopLin.Status.NotMoving AND RightBottomLin.Status.NotMoving THEN	
			GapState:=1;
		END_IF
	1:
		Top_MC_MoveAbsolute.Position:=GapPosition/2;
		Top_MC_MoveAbsolute.Velocity:=GapVelocity/2;
		Bottom_MC_MoveAbsolute.Position:=GapPosition/2;
		Bottom_MC_MoveAbsolute.Velocity:=GapVelocity/2;
		Top_MC_MoveAbsolute.Execute:=TRUE;
		Bottom_MC_MoveAbsolute.Execute:=TRUE;
		fb_ton.IN:=TRUE;
		GapState:=2;
	2:
		(*IF leftTopLin.Status.Moving AND   leftBottomLin.Status.NotMoving THEN (*ÉÏÏÂÁº²»Í¬Ê±¶¯*)
			ErrorID:=3;
			GapState:=-100;
		ELSIF RightTopLin.Status.NotMoving AND RightBottomLin.Status.Moving THEN (*ÉÏÏÂÁº²»Í¬Ê±¶¯*)
			ErrorID:=4;
			GapState:=-100;
		*)
		IF  (LeftTopLin.Status.Moving AND  RightTopLin.Status.NotMoving)
			OR  (LeftTopLin.Status.Moving AND LeftBottomLin.Status.NotMoving)
			OR (LeftTopLin.Status.Moving AND  RightBottomLin.Status.NotMoving)
				OR (RightTopLin.Status.Moving AND  LeftTopLin.Status.NotMoving)
				OR (RightTopLin.Status.Moving AND  LeftBottomLin.Status.NotMoving)
				OR (RightTopLin.Status.Moving AND  RightBottomLin.Status.NotMoving)
					OR (LeftBottomLin.Status.Moving AND  LeftTopLin.Status.NotMoving)
					OR (LeftBottomLin.Status.Moving AND  RightTopLin.Status.NotMoving)
					OR (LeftBottomLin.Status.Moving AND  RightBottomLin.Status.NotMoving)
						OR (RightBottomLin.Status.Moving AND  LeftTopLin.Status.NotMoving)
						OR (RightBottomLin.Status.Moving AND  RightTopLin.Status.NotMoving)
						OR (RightBottomLin.Status.Moving AND  LeftBottomLin.Status.NotMoving) THEN			
			ErrorID:=5;
			GapState:=-100;
		ELSIF NOT Top_MC_MoveAbsolute.Done OR NOT  Bottom_MC_MoveAbsolute.Done THEN		
			(*IF NOT  fb_ton.Q THEN
				GapState:=2;
			ELSE
				ErrorID:=5;
				GapState:=-100;
			END_IF*)
			GapState:=2;
		ELSIF Top_MC_MoveAbsolute.Done  AND  Bottom_MC_MoveAbsolute.Done THEN		
				GapState:=88;
		END_IF
		(*½ÓÊÕµ½stopÐÅºÅÊ±£¬reset×´Ì¬*)
		IF GapReset THEN
			GapState:=89;
		END_IF

	88:
		GapMove:=FALSE;
		GapState:=0;
		GapBusy:=FALSE;
		GapDone:=TRUE;
		Error:=FALSE;
		ErrorID:=0;
		Top_MC_MoveAbsolute.Execute:=FALSE;
		Bottom_MC_MoveAbsolute.Execute:=FALSE;
		fb_ton.IN:=FALSE;
	89:
		GapMove:=FALSE;
		GapState:=0;
		GapBusy:=FALSE;
		GapDone:=FALSE;
		Error:=FALSE;
		ErrorID:=0;
		Top_MC_MoveAbsolute.Execute:=FALSE;
		Bottom_MC_MoveAbsolute.Execute:=FALSE;
		fb_ton.IN:=FALSE;
	99:
		GapMove:=FALSE;
		GapState:=99;
		GapBusy:=FALSE;
		GapDone:=FALSE;
		Error:=TRUE;
		Top_MC_MoveAbsolute.Execute:=FALSE;
		Bottom_MC_MoveAbsolute.Execute:=FALSE;
		fb_ton.IN:=FALSE;
	-100:
		FB_PlcEmergencyStop();
		GapMove:=FALSE;
		GapState:=-100;
		GapBusy:=FALSE;
		GapDone:=FALSE;
		Error:=TRUE;
		Top_MC_MoveAbsolute.Execute:=FALSE;
		Bottom_MC_MoveAbsolute.Execute:=FALSE;
		fb_ton.IN:=FALSE;
END_CASE
END_IF
END_ACTION

ACTION A_LeftBottomMove:
IF LeftBottomMove THEN
LeftBottomBusy:=TRUE;
LeftBottomDone:=FALSE;
fb_ton_debug_3(PT:=t#10s);

IF LeftTopLin.NcToPlc.CoupleState<>0 OR LeftBottomLin.NcToPlc.CoupleState<>0
			OR RightTopLin.NcToPlc.CoupleState<>0 OR RightBottomLin.NcToPlc.CoupleState<>0 THEN
			ErrorID:=1;
			LeftBottomState:=-100;
END_IF
A_MoveMC();
CASE LeftBottomState OF
	0:
		IF Top_MC_MoveAbsolute.Error OR Bottom_MC_MoveAbsolute.Error
			OR RightTopLin_MC_MoveAbsolute.Error OR RightBottomLin_MC_MoveAbsolute.Error THEN	
			ErrorID:=2;
			LeftBottomState:=99;
		ELSIF leftTopLin.Status.NotMoving AND  leftBottomLin.Status.NotMoving
			 AND RightTopLin.Status.NotMoving AND RightBottomLin.Status.NotMoving THEN	
			LeftBottomState:=1;
		END_IF
	1:
		Bottom_MC_MoveAbsolute.Position:=LeftBottomPosition;
		Bottom_MC_MoveAbsolute.Velocity:=LeftBottomVelocity;
		Bottom_MC_MoveAbsolute.Execute:=TRUE;
		fb_ton_debug_3.IN:=TRUE;
		LeftBottomState:=2;
	2:
		IF LeftTopLin.Status.Moving OR RightTopLin.Status.Moving OR RightBottomLin.Status.Moving THEN	
			ErrorID:=3;
			LeftBottomState:=-100;
		ELSIF NOT Bottom_MC_MoveAbsolute.Done THEN		(*ÔË¶¯ÖÐ£¬¼ì²éDoneÐÅºÅ£¬Ã»ÓÐÔòÑ­»·£¬³¬Ê±±¨´í*)
			(*IF NOT  fb_ton.Q THEN
				LeftBottomState:=2;
			ELSE
				ErrorID:=5;
				LeftBottomState:=-100;
			END_IF*)
			LeftBottomState:=2;
		ELSIF Bottom_MC_MoveAbsolute.Done THEN		
				LeftBottomState:=88;
		END_IF

		IF LeftBottomReset THEN
			LeftBottomState:=89;
		END_IF

	88:
		LeftBottomMove:=FALSE;
		LeftBottomState:=0;
		LeftBottomBusy:=FALSE;
		LeftBottomDone:=TRUE;
		Error:=FALSE;
		ErrorID:=0;
		Bottom_MC_MoveAbsolute.Execute:=FALSE;
		fb_ton_debug_3.IN:=FALSE;
	89:
		LeftBottomMove:=FALSE;
		LeftBottomState:=0;
		LeftBottomBusy:=FALSE;
		LeftBottomDone:=FALSE;
		Error:=FALSE;
		ErrorID:=0;
		Bottom_MC_MoveAbsolute.Execute:=FALSE;
		fb_ton_debug_3.IN:=FALSE;
	99:
		LeftBottomMove:=FALSE;
		LeftBottomState:=99;
		LeftBottomBusy:=FALSE;
		LeftBottomDone:=FALSE;
		Error:=TRUE;
		Bottom_MC_MoveAbsolute.Execute:=FALSE;
		fb_ton_debug_3.IN:=FALSE;
	-100:
		FB_PlcEmergencyStop();
		LeftBottomMove:=FALSE;
		LeftBottomState:=-100;
		LeftBottomBusy:=FALSE;
		LeftBottomDone:=FALSE;
		Error:=TRUE;
		Bottom_MC_MoveAbsolute.Execute:=FALSE;
		fb_ton_debug_3.IN:=FALSE;
END_CASE
END_IF
END_ACTION

ACTION A_LeftTopMove:
IF LeftTopMove THEN
LeftTopBusy:=TRUE;
LeftTopDone:=FALSE;
fb_ton_debug_1(PT:=t#10s);

IF LeftTopLin.NcToPlc.CoupleState<>0 OR LeftBottomLin.NcToPlc.CoupleState<>0
			OR RightTopLin.NcToPlc.CoupleState<>0 OR RightBottomLin.NcToPlc.CoupleState<>0 THEN
			ErrorID:=1;
			LeftTopState:=-100;
END_IF
A_MoveMC();
CASE LeftTopState OF
	0:
		IF Top_MC_MoveAbsolute.Error OR Bottom_MC_MoveAbsolute.Error
			OR RightTopLin_MC_MoveAbsolute.Error OR RightBottomLin_MC_MoveAbsolute.Error THEN		
			ErrorID:=2;
			LeftTopState:=99;
		ELSIF leftTopLin.Status.NotMoving AND  leftBottomLin.Status.NotMoving
			 AND RightTopLin.Status.NotMoving AND RightBottomLin.Status.NotMoving THEN
			LeftTopState:=1;
		END_IF
	1:
		Top_MC_MoveAbsolute.Position:=LeftTopPosition;
		Top_MC_MoveAbsolute.Velocity:=LeftTopVelocity;
		Top_MC_MoveAbsolute.Execute:=TRUE;
		fb_ton_debug_1.IN:=TRUE;
		LeftTopState:=2;
	2:
		IF RightTopLin.Status.Moving OR LeftBottomLin.Status.Moving OR RightBottomLin.Status.Moving THEN
			ErrorID:=3;
			LeftTopState:=-100;
		ELSIF NOT Top_MC_MoveAbsolute.Done THEN	
			(*IF NOT  fb_ton.Q THEN
				LeftTopState:=2;
			ELSE
				ErrorID:=5;
				LeftTopState:=-100;
			END_IF*)
			LeftTopState:=2;
		ELSIF Top_MC_MoveAbsolute.Done THEN		
				LeftTopState:=88;
		END_IF
		(*½ÓÊÕµ½stopÐÅºÅÊ±£¬reset×´Ì¬*)
		IF LeftTopReset THEN
			LeftTopState:=89;
		END_IF

	88:
		LeftTopMove:=FALSE;
		LeftTopState:=0;
		LeftTopBusy:=FALSE;
		LeftTopDone:=TRUE;
		Error:=FALSE;
		ErrorID:=0;
		Top_MC_MoveAbsolute.Execute:=FALSE;
		fb_ton_debug_1.IN:=FALSE;
	89:
		LeftTopMove:=FALSE;
		LeftTopState:=0;
		LeftTopBusy:=FALSE;
		LeftTopDone:=FALSE;
		Error:=FALSE;
		ErrorID:=0;
		Top_MC_MoveAbsolute.Execute:=FALSE;
		fb_ton_debug_1.IN:=FALSE;
	99:
		LeftTopMove:=FALSE;
		LeftTopState:=99;
		LeftTopBusy:=FALSE;
		LeftTopDone:=FALSE;
		Error:=TRUE;
		Top_MC_MoveAbsolute.Execute:=FALSE;
		fb_ton_debug_1.IN:=FALSE;
	-100:
		FB_PlcEmergencyStop();
		LeftTopMove:=FALSE;
		LeftTopState:=-100;
		LeftTopBusy:=FALSE;
		LeftTopDone:=FALSE;
		Error:=TRUE;
		Top_MC_MoveAbsolute.Execute:=FALSE;
		fb_ton_debug_1.IN:=FALSE;
END_CASE
END_IF
END_ACTION

ACTION A_MoveMC:
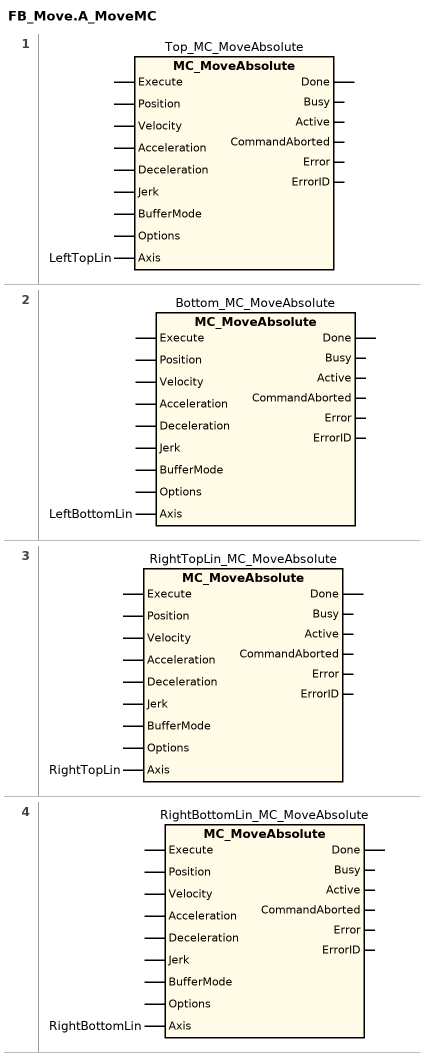
// NETWORK 1
Top_MC_MoveAbsolute(Axis := LeftTopLin); // MC_MoveAbsolute

// NETWORK 2
Bottom_MC_MoveAbsolute(Axis := LeftBottomLin); // MC_MoveAbsolute

// NETWORK 3
RightTopLin_MC_MoveAbsolute(Axis := RightTopLin); // MC_MoveAbsolute

// NETWORK 4
RightBottomLin_MC_MoveAbsolute(Axis := RightBottomLin); // MC_MoveAbsolute
END_ACTION

ACTION A_RightBottomMove:
IF RightBottomMove THEN
RightBottomBusy:=TRUE;
RightBottomDone:=FALSE;
fb_ton_debug_4(PT:=t#10s);

IF LeftTopLin.NcToPlc.CoupleState<>0 OR LeftBottomLin.NcToPlc.CoupleState<>0
			OR RightTopLin.NcToPlc.CoupleState<>0 OR RightBottomLin.NcToPlc.CoupleState<>0 THEN
			ErrorID:=1;
			RightBottomState:=-100;
END_IF
A_MoveMC();
CASE RightBottomState OF
	0:
		IF Top_MC_MoveAbsolute.Error OR Bottom_MC_MoveAbsolute.Error
			OR RightTopLin_MC_MoveAbsolute.Error OR RightBottomLin_MC_MoveAbsolute.Error THEN		
			ErrorID:=2;
			RightBottomState:=99;
		ELSIF leftTopLin.Status.NotMoving AND  leftBottomLin.Status.NotMoving
			 AND RightTopLin.Status.NotMoving AND RightBottomLin.Status.NotMoving THEN	
			RightBottomState:=1;
		END_IF
	1:
		RightBottomLin_MC_MoveAbsolute.Position:=RightBottomPosition;
		RightBottomLin_MC_MoveAbsolute.Velocity:=RightBottomVelocity;
		RightBottomLin_MC_MoveAbsolute.Execute:=TRUE;
		fb_ton_debug_4.IN:=TRUE;
		RightBottomState:=2;
	2:
		IF LeftTopLin.Status.Moving OR RightTopLin.Status.Moving  OR LeftBottomLin.Status.Moving THEN	
			ErrorID:=3;
			RightBottomState:=-100;
		ELSIF NOT RightBottomLin_MC_MoveAbsolute.Done THEN	
			(*IF NOT  fb_ton.Q THEN
				LeftTopState:=2;
			ELSE
				ErrorID:=5;
				LeftTopState:=-100;
			END_IF*)
			RightBottomState:=2;
		ELSIF RightBottomLin_MC_MoveAbsolute.Done THEN		
				RightBottomState:=88;
		END_IF
		(*½ÓÊÕµ½stopÐÅºÅÊ±£¬reset×´Ì¬*)
		IF RightBottomReset THEN
			RightBottomState:=89;
		END_IF

	88:
		RightBottomMove:=FALSE;
		RightBottomState:=0;
		RightBottomBusy:=FALSE;
		RightBottomDone:=TRUE;
		Error:=FALSE;
		ErrorID:=0;
		RightBottomLin_MC_MoveAbsolute.Execute:=FALSE;
		fb_ton_debug_4.IN:=FALSE;
	89:
		RightBottomMove:=FALSE;
		RightBottomState:=0;
		RightBottomBusy:=FALSE;
		RightBottomDone:=FALSE;
		Error:=FALSE;
		ErrorID:=0;
		RightBottomLin_MC_MoveAbsolute.Execute:=FALSE;
		fb_ton_debug_4.IN:=FALSE;
	99:
		RightBottomMove:=FALSE;
		RightBottomState:=99;
		RightBottomBusy:=FALSE;
		RightBottomDone:=FALSE;
		Error:=TRUE;
		RightBottomLin_MC_MoveAbsolute.Execute:=FALSE;
		fb_ton_debug_4.IN:=FALSE;
	-100:
		FB_PlcEmergencyStop();
		RightBottomMove:=FALSE;
		RightBottomState:=-100;
		RightBottomBusy:=FALSE;
		RightBottomDone:=FALSE;
		Error:=TRUE;
		RightBottomLin_MC_MoveAbsolute.Execute:=FALSE;
		fb_ton_debug_4.IN:=FALSE;
END_CASE
END_IF
END_ACTION

ACTION A_RightTopMove:
IF RightTopMove THEN
RightTopBusy:=TRUE;
RightTopDone:=FALSE;
fb_ton_debug_2(PT:=t#10s);

IF LeftTopLin.NcToPlc.CoupleState<>0 OR LeftBottomLin.NcToPlc.CoupleState<>0
			OR RightTopLin.NcToPlc.CoupleState<>0 OR RightBottomLin.NcToPlc.CoupleState<>0 THEN
			ErrorID:=1;
			RightTopState:=-100;
END_IF
A_MoveMC();
CASE RightTopState OF
	0:
		IF Top_MC_MoveAbsolute.Error OR Bottom_MC_MoveAbsolute.Error
			OR RightTopLin_MC_MoveAbsolute.Error OR RightBottomLin_MC_MoveAbsolute.Error THEN
			ErrorID:=2;
			RightTopState:=99;
		ELSIF leftTopLin.Status.NotMoving AND  leftBottomLin.Status.NotMoving
			 AND RightTopLin.Status.NotMoving AND RightBottomLin.Status.NotMoving THEN
			RightTopState:=1;
		END_IF
	1:
		RightTopLin_MC_MoveAbsolute.Position:=RightTopPosition;
		RightTopLin_MC_MoveAbsolute.Velocity:=RightTopVelocity;
		RightTopLin_MC_MoveAbsolute.Execute:=TRUE;
		fb_ton_debug_2.IN:=TRUE;
		RightTopState:=2;
	2:
		IF LeftTopLin.Status.Moving OR LeftBottomLin.Status.Moving OR RightBottomLin.Status.Moving THEN	
			ErrorID:=3;
			RightTopState:=-100;
		ELSIF NOT RightTopLin_MC_MoveAbsolute.Done THEN	
			(*IF NOT  fb_ton.Q THEN
				LeftTopState:=2;
			ELSE
				ErrorID:=5;
				LeftTopState:=-100;
			END_IF*)
			RightTopState:=2;
		ELSIF RightTopLin_MC_MoveAbsolute.Done THEN	
				RightTopState:=88;
		END_IF
		(*½ÓÊÕµ½stopÐÅºÅÊ±£¬reset×´Ì¬*)
		IF RightTopReset THEN
			RightTopState:=89;
		END_IF

	88:
		RightTopMove:=FALSE;
		RightTopState:=0;
		RightTopBusy:=FALSE;
		RightTopDone:=TRUE;
		Error:=FALSE;
		ErrorID:=0;
		RightTopLin_MC_MoveAbsolute.Execute:=FALSE;
		fb_ton_debug_2.IN:=FALSE;
	89:
		RightTopMove:=FALSE;
		RightTopState:=0;
		RightTopBusy:=FALSE;
		RightTopDone:=FALSE;
		Error:=FALSE;
		ErrorID:=0;
		RightTopLin_MC_MoveAbsolute.Execute:=FALSE;
		fb_ton_debug_2.IN:=FALSE;
	99:
		RightTopMove:=FALSE;
		RightTopState:=99;
		RightTopBusy:=FALSE;
		RightTopDone:=FALSE;
		Error:=TRUE;
		RightTopLin_MC_MoveAbsolute.Execute:=FALSE;
		fb_ton_debug_2.IN:=FALSE;
	-100:
		FB_PlcEmergencyStop();
		RightTopMove:=FALSE;
		RightTopState:=-100;
		RightTopBusy:=FALSE;
		RightTopDone:=FALSE;
		Error:=TRUE;
		RightTopLin_MC_MoveAbsolute.Execute:=FALSE;
		fb_ton_debug_2.IN:=FALSE;
END_CASE
END_IF
END_ACTION

ACTION A_TaperMove:
IF TaperMove THEN
TaperBusy:=TRUE;
TaperDone:=FALSE;
fb_ton(PT:=t#80s);

IF LeftTopLin.NcToPlc.CoupleState<>0 OR LeftBottomLin.NcToPlc.CoupleState<>0
			OR RightTopLin.NcToPlc.CoupleState<>0 OR RightBottomLin.NcToPlc.CoupleState<>0 THEN
			ErrorID:=1;
			TaperState:=-100;
END_IF

IF LeftTopLin.Status.Moving OR LeftBottomLin.Status.Moving THEN
			ErrorID:=2;
			TaperState:=-100;
END_IF

IF (RightTopLin.Status.Moving AND RightBottomLin.Status.NotMoving) OR (RightTopLin.Status.NotMoving AND RightBottomLin.Status.Moving) THEN
			ErrorID:=3;
			TaperState:=-100;
END_IF
A_MoveMC();
CASE TaperState OF

	0:
		IF RightTopLin.Status.Moving OR RightBottomLin.Status.Moving THEN	
			TaperState:=88;
		ELSIF Top_MC_MoveAbsolute.Error OR Bottom_MC_MoveAbsolute.Error THEN	
			ErrorID:=4;
			TaperState:=99;
		ELSIF leftTopLin.Status.NotMoving AND  leftBottomLin.Status.NotMoving
			 AND RightTopLin.Status.NotMoving AND RightBottomLin.Status.NotMoving THEN
			TaperState:=1;
		END_IF
	1:
		RightTopLin_MC_MoveAbsolute.Position:=TaperPosition;
		RightTopLin_MC_MoveAbsolute.Velocity:=TaperVelocity;
		RightBottomLin_MC_MoveAbsolute.Position:=TaperPosition;
		RightBottomLin_MC_MoveAbsolute.Velocity:=TaperVelocity;
		RightTopLin_MC_MoveAbsolute.Execute:=TRUE;
		RightBottomLin_MC_MoveAbsolute.Execute:=TRUE;
		fb_ton.IN:=TRUE;
		TaperState:=2;
	2:
		IF leftTopLin.Status.Moving OR   leftBottomLin.Status.Moving THEN		
			ErrorID:=5;
			TaperState:=-100;
		ELSIF  (RightTopLin.Status.Moving AND RightBottomLin.Status.NotMoving) OR (RightTopLin.Status.NotMoving AND RightBottomLin.Status.Moving) THEN
			ErrorID:=6;
			TaperState:=-100;
		ELSIF NOT RightTopLin_MC_MoveAbsolute.Done OR NOT  RightBottomLin_MC_MoveAbsolute.Done THEN		
			(*IF NOT  fb_ton.Q THEN
				TaperState:=2;
			ELSE
				ErrorID:=5;
				TaperState:=-100;
			END_IF*)
			TaperState:=2;
		ELSIF RightTopLin_MC_MoveAbsolute.Done  AND  RightBottomLin_MC_MoveAbsolute.Done THEN	
				TaperState:=88;
		END_IF

		IF TaperReset THEN
			TaperState:=89;
		END_IF

	88:
		TaperMove:=FALSE;
		TaperState:=0;
		TaperBusy:=FALSE;
		TaperDone:=TRUE;
		Error:=FALSE;
		ErrorID:=0;
		RightTopLin_MC_MoveAbsolute.Execute:=FALSE;
		RightBottomLin_MC_MoveAbsolute.Execute:=FALSE;
		fb_ton.IN:=FALSE;
	89:
		TaperMove:=FALSE;
		TaperState:=0;
		TaperBusy:=FALSE;
		TaperDone:=FALSE;
		Error:=FALSE;
		ErrorID:=0;
		RightTopLin_MC_MoveAbsolute.Execute:=FALSE;
		RightBottomLin_MC_MoveAbsolute.Execute:=FALSE;
		fb_ton.IN:=FALSE;
	99:
		TaperMove:=FALSE;
		TaperState:=99;
		TaperBusy:=FALSE;
		TaperDone:=FALSE;
		Error:=TRUE;
		RightTopLin_MC_MoveAbsolute.Execute:=FALSE;
		RightBottomLin_MC_MoveAbsolute.Execute:=FALSE;
		fb_ton.IN:=FALSE;
	-100:
		FB_PlcEmergencyStop();
		TaperMove:=FALSE;
		TaperState:=-100;
		TaperBusy:=FALSE;
		TaperDone:=FALSE;
		Error:=TRUE;
		RightTopLin_MC_MoveAbsolute.Execute:=FALSE;
		RightBottomLin_MC_MoveAbsolute.Execute:=FALSE;
		fb_ton.IN:=FALSE;
END_CASE
END_IF
END_ACTION

ACTION A_TopMove:
IF TopMove THEN
TopBusy:=TRUE;
TopDone:=FALSE;
fb_ton1(PT:=T#80S);(*2mm/s max spees,120mm*)
A_MoveMC();
CASE TopState OF
	0:
		IF Top_MC_MoveAbsolute.Error OR RightTopLin_MC_MoveAbsolute.Error THEN		
			ErrorID:=2;
			TopState:=99;
		END_IF
		TopState:=1;
	1:
		Top_MC_MoveAbsolute.Position:=TopPosition;
		Top_MC_MoveAbsolute.Velocity:=TopVelocity;
		Top_MC_MoveAbsolute.Execute:=TRUE;
		RightTopLin_MC_MoveAbsolute.Position:=TopPosition;
		RightTopLin_MC_MoveAbsolute.Velocity:=TopVelocity;
		RightTopLin_MC_MoveAbsolute.Execute:=TRUE;
		fb_ton1.IN:=TRUE;
		TopState:=2;
	2:
		IF leftBottomLin.Status.Moving OR RightBottomLin.Status.Moving THEN	
			ErrorID:=3;
			TopState:=-100;
		ELSIF  (LeftTopLin.Status.Moving AND  RightTopLin.Status.NotMoving)
				OR (RightTopLin.Status.Moving AND  LeftTopLin.Status.NotMoving) THEN			
			//ErrorID:=4;
			//TopState:=-100;
		ELSIF NOT Top_MC_MoveAbsolute.Done OR NOT RightTopLin_MC_MoveAbsolute.Done THEN		
			TopState:=2;
		ELSIF Top_MC_MoveAbsolute.Done AND RightTopLin_MC_MoveAbsolute.Done THEN		
				TopState:=88;
		END_IF
		(*½ÓÊÕµ½stopÐÅºÅÊ±£¬reset×´Ì¬*)
		IF TopReset THEN
			TopState:=89;
		END_IF

	88:
		TopMove:=FALSE;
		TopState:=0;
		TopBusy:=FALSE;
		TopDone:=TRUE;
		Error:=FALSE;
		ErrorID:=0;
		Top_MC_MoveAbsolute.Execute:=FALSE;
		RightTopLin_MC_MoveAbsolute.Execute:=FALSE;
		fb_ton1.IN:=FALSE;
	89:
		TopMove:=FALSE;
		TopState:=0;
		TopBusy:=FALSE;
		TopDone:=FALSE;
		Error:=FALSE;
		ErrorID:=0;
		Top_MC_MoveAbsolute.Execute:=FALSE;
		RightTopLin_MC_MoveAbsolute.Execute:=FALSE;
		fb_ton1.IN:=FALSE;
	99:
		TopMove:=FALSE;
		TopState:=99;
		TopBusy:=FALSE;
		TopDone:=FALSE;
		Error:=TRUE;
		Top_MC_MoveAbsolute.Execute:=FALSE;
		RightTopLin_MC_MoveAbsolute.Execute:=FALSE;
		fb_ton1.IN:=FALSE;
	-100:
		FB_PlcEmergencyStop();
		TopMove:=FALSE;
		TopState:=-100;
		TopBusy:=FALSE;
		TopDone:=FALSE;
		Error:=TRUE;
		Top_MC_MoveAbsolute.Execute:=FALSE;
		RightTopLin_MC_MoveAbsolute.Execute:=FALSE;
		fb_ton1.IN:=FALSE;
END_CASE
END_IF
END_ACTION

END_FUNCTION_BLOCK

// ---- POUs/CommonFB/MainFB/FB_Stop.TcPOU
FUNCTION_BLOCK FB_Stop
VAR_INPUT
(*È«¾Ö*)
	Mode:DINT;
	PowerState:DINT;
	CoupleState:DINT;
	(*GapMode*)
	GapStop:BOOL;
	(*BCGapMode*)
	BCGapStop:BOOL;
	(*SingleCarrierMode*)
	TopStop:BOOL;
	BottomStop:BOOL;
	(*TaperMode*)
	TaperStop:BOOL;
	(*DebugMode*)
	LeftTopStop:BOOL;
	RightTopStop:BOOL;
	LeftBottomStop:BOOL;
	RightBottomStop:BOOL;
END_VAR
VAR_OUTPUT
	FbID:DINT:=1001;
	GapState:DINT;
	GapBusy:BOOL;
	GapDone:BOOL;

	BCGapState:DINT;
	BCGapBusy:BOOL;
	BCGapDone:BOOL;

	TopState:DINT;
	TopBusy:BOOL;
	TopDone:BOOL;
	BottomState:DINT;
	BottomBusy:BOOL;
	BottomDone:BOOL;

	TaperState:DINT;
	TaperBusy:BOOL;
	TaperDone:BOOL;

	LeftTopState:DINT;
	LeftTopBusy:BOOL;
	LeftTopDone:BOOL;
	RightTopState:DINT;
	RightTopBusy:BOOL;
	RightTopDone:BOOL;
	LeftBottomState:DINT;
	LeftBottomBusy:BOOL;
	LeftBottomDone:BOOL;
	RightBottomState:DINT;
	RightBottomBusy:BOOL;
	RightBottomDone:BOOL;

	Error:BOOL;
	ErrorID:DINT;
END_VAR
VAR
	Top_MC_Stop: MC_Stop;
	Bottom_MC_Stop: MC_Stop;
	RightTopLin_MC_Stop: MC_Stop;
	RightBottomLin_MC_Stop: MC_Stop;
	fb_ton: TON;
	fb_ton1: TON;
	fb_ton2: TON;
	fb_ton_debug_1:TON;
	fb_ton_debug_2:TON;
	fb_ton_debug_3:TON;
	fb_ton_debug_4:TON;
	fb_ton_BC: TON;
END_VAR

IF PowerState=1 THEN
	IF Mode=1 AND CoupleState=1 THEN
		A_GapStop();
	ELSIF Mode=2 AND CoupleState=0 AND TopStop THEN
		A_TopStop();
	ELSIF Mode=2 AND CoupleState=0 AND BottomStop THEN
		A_BottomStop();
	ELSIF Mode=3 AND CoupleState=0 AND TaperStop THEN
		A_TaperStop();
	ELSIF Mode=4 AND CoupleState=0 AND LeftTopStop THEN
		A_LeftTopStop();
	ELSIF Mode=4 AND CoupleState=0 AND RightTopStop THEN
		A_RightTopStop();
	ELSIF Mode=4 AND CoupleState=0 AND LeftBottomStop THEN
		A_LeftBottomStop();
	ELSIF Mode=4 AND CoupleState=0 AND RightBottomStop THEN
		A_RightBottomStop();
	ELSIF Mode=5 AND CoupleState=0 AND BCGapStop THEN
		A_BCGapStop();
	ELSE
		FB_PlcEmergencyStop();
	END_IF
END_IF

ACTION A_BCGapStop:
IF BCGapStop THEN
BCGapBusy:=TRUE;
BCGapDone:=FALSE;
fb_ton_BC(PT:=t#100ms);
A_StopMC();
CASE BCGapState OF
	0:
		IF Top_MC_Stop.Error OR Bottom_MC_Stop.Error OR RightTopLin_MC_Stop.Error OR RightBottomLin_MC_Stop.Error THEN
			ErrorID:=1;
			BCGapState:=-100;
			Top_MC_Stop.Execute:=FALSE;
			Bottom_MC_Stop.Execute:=FALSE;
			RightTopLin_MC_Stop.Execute:=FALSE;
			RightBottomLin_MC_Stop.Execute:=FALSE;
			A_StopMC();
		ELSE
			BCGapState:=1;
		END_IF
	1:
		Top_MC_Stop.Execute:=TRUE;
		Bottom_MC_Stop.Execute:=TRUE;
		RightTopLin_MC_Stop.Execute:=TRUE;
		RightBottomLin_MC_Stop.Execute:=TRUE;
		fb_ton_BC.IN:=TRUE;
		BCGapState:=2;
	2:
		IF  NOT Top_MC_Stop.Done OR NOT Bottom_MC_Stop.Done OR NOT RightTopLin_MC_Stop.Done OR NOT RightBottomLin_MC_Stop.Done THEN
				BCGapState:=2;
		ELSE
			BCGapState:=88;
			Top_MC_Stop.Execute:=FALSE;
			Bottom_MC_Stop.Execute:=FALSE;
			RightTopLin_MC_Stop.Execute:=FALSE;
			RightBottomLin_MC_Stop.Execute:=FALSE;
			A_StopMC();
		END_IF

	88:
		BCGapStop:=FALSE;
		BCGapState:=0;
		BCGapBusy:=FALSE;
		BCGapDone:=TRUE;
		Error:=FALSE;
		ErrorID:=0;
		fb_ton_BC.IN:=FALSE;

	-100:
		FB_PlcEmergencyStop();
		BCGapStop:=FALSE;
		BCGapState:=-100;
		BCGapBusy:=FALSE;
		BCGapDone:=FALSE;
		Error:=TRUE;
		Top_MC_Stop.Execute:=FALSE;
		Bottom_MC_Stop.Execute:=FALSE;
		RightTopLin_MC_Stop.Execute:=FALSE;
		RightBottomLin_MC_Stop.Execute:=FALSE;
		A_StopMC();
		fb_ton_BC.IN:=FALSE;

END_CASE
END_IF
END_ACTION

ACTION A_BottomStop:
IF BottomStop THEN
BottomBusy:=TRUE;
BottomDone:=FALSE;
fb_ton2(PT:=t#100ms);
A_StopMC();
CASE BottomState OF
	0:
		IF Bottom_MC_Stop.Error OR RightBottomLin_MC_Stop.Error THEN
			ErrorID:=1;
			BottomState:=-100;
			Bottom_MC_Stop.Execute:=FALSE;
			RightBottomLin_MC_Stop.Execute:=FALSE;
			A_StopMC();
		ELSE
			BottomState:=1;
		END_IF
	1:
		Bottom_MC_Stop.Execute:=TRUE;
		RightBottomLin_MC_Stop.Execute:=TRUE;
		fb_ton2.IN:=TRUE;
		BottomState:=2;
	2:
		IF  NOT Bottom_MC_Stop.Done OR NOT Bottom_MC_Stop.Done THEN
				BottomState:=2;
		ELSE
			BottomState:=88;
			Bottom_MC_Stop.Execute:=FALSE;
			RightBottomLin_MC_Stop.Execute:=FALSE;
			A_StopMC();
		END_IF

	88:
		BottomStop:=FALSE;
		BottomState:=0;
		BottomBusy:=FALSE;
		BottomDone:=TRUE;
		Error:=FALSE;
		ErrorID:=0;
		fb_ton2.IN:=FALSE;

	-100:
		FB_PlcEmergencyStop();
		BottomStop:=FALSE;
		BottomState:=-100;
		BottomBusy:=FALSE;
		BottomDone:=FALSE;
		Error:=TRUE;
		Bottom_MC_Stop.Execute:=FALSE;
		RightBottomLin_MC_Stop.Execute:=FALSE;
		A_StopMC();
		fb_ton2.IN:=FALSE;

END_CASE
END_IF
END_ACTION

ACTION A_GapStop:
IF GapStop THEN
GapBusy:=TRUE;
GapDone:=FALSE;
fb_ton(PT:=t#100ms);
A_StopMC();
CASE GapState OF
	0:
		IF Top_MC_Stop.Error OR Bottom_MC_Stop.Error THEN
			ErrorID:=1;
			GapState:=-100;
			Top_MC_Stop.Execute:=FALSE;
			Bottom_MC_Stop.Execute:=FALSE;
			A_StopMC();
		ELSE
			GapState:=1;
		END_IF
	1:
		Top_MC_Stop.Execute:=TRUE;
		Bottom_MC_Stop.Execute:=TRUE;
		fb_ton.IN:=TRUE;
		GapState:=2;
	2:
		IF  NOT Top_MC_Stop.Done OR NOT Bottom_MC_Stop.Done THEN
				GapState:=2;
		ELSE
			GapState:=88;
			Top_MC_Stop.Execute:=FALSE;
			Bottom_MC_Stop.Execute:=FALSE;
			A_StopMC();
		END_IF

	88:
		GapStop:=FALSE;
		GapState:=0;
		GapBusy:=FALSE;
		GapDone:=TRUE;
		Error:=FALSE;
		ErrorID:=0;
		fb_ton.IN:=FALSE;

	-100:
		FB_PlcEmergencyStop();
		GapStop:=FALSE;
		GapState:=-100;
		GapBusy:=FALSE;
		GapDone:=FALSE;
		Error:=TRUE;
		Top_MC_Stop.Execute:=FALSE;
		Bottom_MC_Stop.Execute:=FALSE;
		A_StopMC();
		fb_ton.IN:=FALSE;

END_CASE
END_IF
END_ACTION

ACTION A_LeftBottomStop:
IF LeftBottomStop THEN
LeftBottomBusy:=TRUE;
LeftBottomDone:=FALSE;
fb_ton_debug_3(PT:=t#100ms);
A_StopMC();
CASE LeftBottomState OF
	0:
		IF Bottom_MC_Stop.Error THEN
			ErrorID:=41;
			LeftBottomState:=-100;
			Bottom_MC_Stop.Execute:=FALSE;
			A_StopMC();
		ELSE
			LeftBottomState:=1;
		END_IF
	1:
		Bottom_MC_Stop.Execute:=TRUE;
		fb_ton_debug_3.IN:=TRUE;
		LeftBottomState:=2;
	2:
		IF  NOT Bottom_MC_Stop.Done THEN
				LeftBottomState:=2;
		ELSE
			LeftBottomState:=88;
			Bottom_MC_Stop.Execute:=FALSE;
			A_StopMC();
		END_IF

	88:
		LeftBottomStop:=FALSE;
		LeftBottomState:=0;
		LeftBottomBusy:=FALSE;
		LeftBottomDone:=TRUE;
		Error:=FALSE;
		ErrorID:=0;
		fb_ton_debug_3.IN:=FALSE;

	-100:
		FB_PlcEmergencyStop();
		LeftBottomStop:=FALSE;
		LeftBottomState:=-100;
		LeftBottomBusy:=FALSE;
		LeftBottomDone:=FALSE;
		Error:=TRUE;
		Bottom_MC_Stop.Execute:=FALSE;
		A_StopMC();
		fb_ton_debug_3.IN:=FALSE;

END_CASE
END_IF
END_ACTION

ACTION A_LeftTopStop:
IF LeftTopStop THEN
LeftTopBusy:=TRUE;
LeftTopDone:=FALSE;
fb_ton_debug_1(PT:=t#100ms);
A_StopMC();
CASE LeftTopState OF
	0:
		IF Top_MC_Stop.Error THEN
			ErrorID:=41;
			LeftTopState:=-100;
			Top_MC_Stop.Execute:=FALSE;
			A_StopMC();
		ELSE
			LeftTopState:=1;
		END_IF
	1:
		Top_MC_Stop.Execute:=TRUE;
		fb_ton_debug_1.IN:=TRUE;
		LeftTopState:=2;
	2:
		IF  NOT Top_MC_Stop.Done THEN
				LeftTopState:=2;
		ELSE
			LeftTopState:=88;
			Top_MC_Stop.Execute:=FALSE;
			A_StopMC();
		END_IF

	88:
		LeftTopStop:=FALSE;
		LeftTopState:=0;
		LeftTopBusy:=FALSE;
		LeftTopDone:=TRUE;
		Error:=FALSE;
		ErrorID:=0;
		fb_ton_debug_1.IN:=FALSE;

	-100:
		FB_PlcEmergencyStop();
		LeftTopStop:=FALSE;
		LeftTopState:=-100;
		LeftTopBusy:=FALSE;
		LeftTopDone:=FALSE;
		Error:=TRUE;
		Top_MC_Stop.Execute:=FALSE;
		A_StopMC();
		fb_ton_debug_1.IN:=FALSE;

END_CASE
END_IF
END_ACTION

ACTION A_RightBottomStop:
IF RightBottomStop THEN
RightBottomBusy:=TRUE;
RightBottomDone:=FALSE;
fb_ton_debug_4(PT:=t#100ms);
A_StopMC();
CASE RightBottomState OF
	0:
		IF RightBottomLin_MC_Stop.Error THEN
			ErrorID:=41;
			RightBottomState:=-100;
			RightBottomLin_MC_Stop.Execute:=FALSE;
			A_StopMC();
		ELSE
			RightBottomState:=1;
		END_IF
	1:
		RightBottomLin_MC_Stop.Execute:=TRUE;
		fb_ton_debug_4.IN:=TRUE;
		RightBottomState:=2;
	2:
		IF  NOT RightBottomLin_MC_Stop.Done THEN
				RightBottomState:=2;
		ELSE
			RightBottomState:=88;
			RightBottomLin_MC_Stop.Execute:=FALSE;
			A_StopMC();
		END_IF

	88:
		RightBottomStop:=FALSE;
		RightBottomState:=0;
		RightBottomBusy:=FALSE;
		RightBottomDone:=TRUE;
		Error:=FALSE;
		ErrorID:=0;
		fb_ton_debug_4.IN:=FALSE;

	-100:
		FB_PlcEmergencyStop();
		RightBottomStop:=FALSE;
		RightBottomState:=-100;
		RightBottomBusy:=FALSE;
		RightBottomDone:=FALSE;
		Error:=TRUE;
		RightBottomLin_MC_Stop.Execute:=FALSE;
		A_StopMC();
		fb_ton_debug_4.IN:=FALSE;

END_CASE
END_IF
END_ACTION

ACTION A_RightTopStop:
IF RightTopStop THEN
RightTopBusy:=TRUE;
RightTopDone:=FALSE;
fb_ton_debug_2(PT:=t#100ms);
A_StopMC();
CASE RightTopState OF
	0:
		IF RightTopLin_MC_Stop.Error THEN
			ErrorID:=41;
			RightTopState:=-100;
			RightTopLin_MC_Stop.Execute:=FALSE;
			A_StopMC();
		ELSE
			RightTopState:=1;
		END_IF
	1:
		RightTopLin_MC_Stop.Execute:=TRUE;
		fb_ton_debug_2.IN:=TRUE;
		RightTopState:=2;
	2:
		IF  NOT RightTopLin_MC_Stop.Done THEN
				RightTopState:=2;
		ELSE
			RightTopState:=88;
			RightTopLin_MC_Stop.Execute:=FALSE;
			A_StopMC();
		END_IF

	88:
		RightTopStop:=FALSE;
		RightTopState:=0;
		RightTopBusy:=FALSE;
		RightTopDone:=TRUE;
		Error:=FALSE;
		ErrorID:=0;
		fb_ton_debug_2.IN:=FALSE;

	-100:
		FB_PlcEmergencyStop();
		RightTopStop:=FALSE;
		RightTopState:=-100;
		RightTopBusy:=FALSE;
		RightTopDone:=FALSE;
		Error:=TRUE;
		RightTopLin_MC_Stop.Execute:=FALSE;
		A_StopMC();
		fb_ton_debug_2.IN:=FALSE;

END_CASE
END_IF
END_ACTION

ACTION A_StopMC:
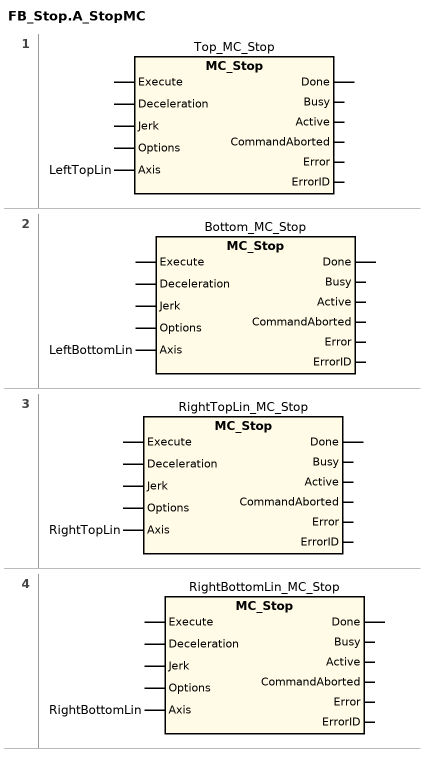
// NETWORK 1
Top_MC_Stop(Axis := LeftTopLin); // MC_Stop

// NETWORK 2
Bottom_MC_Stop(Axis := LeftBottomLin); // MC_Stop

// NETWORK 3
RightTopLin_MC_Stop(Axis := RightTopLin); // MC_Stop

// NETWORK 4
RightBottomLin_MC_Stop(Axis := RightBottomLin); // MC_Stop
END_ACTION

ACTION A_TaperStop:
IF TaperStop THEN
TaperBusy:=TRUE;
TaperDone:=FALSE;
fb_ton(PT:=t#100ms);
A_StopMC();
CASE TaperState OF
	0:
		IF RightTopLin_MC_Stop.Error  OR RightBottomLin_MC_Stop.Error THEN
			ErrorID:=1;
			TaperState:=-100;
			RightTopLin_MC_Stop.Execute:=FALSE;
			RightBottomLin_MC_Stop.Execute:=FALSE;
			A_StopMC();
		ELSE
			TaperState:=1;
		END_IF
	1:
		RightTopLin_MC_Stop.Execute:=TRUE;
		RightBottomLin_MC_Stop.Execute:=TRUE;
		fb_ton.IN:=TRUE;
		TaperState:=2;
	2:
		IF  NOT RightTopLin_MC_Stop.Done OR NOT RightBottomLin_MC_Stop.Done THEN
				TaperState:=2;
		ELSE
			TaperState:=88;
			RightTopLin_MC_Stop.Execute:=FALSE;
			RightBottomLin_MC_Stop.Execute:=FALSE;
			A_StopMC();
		END_IF

	88:
		TaperStop:=FALSE;
		TaperState:=0;
		TaperBusy:=FALSE;
		TaperDone:=TRUE;
		Error:=FALSE;
		ErrorID:=0;
		fb_ton.IN:=FALSE;

	-100:
		FB_PlcEmergencyStop();
		TaperStop:=FALSE;
		TaperState:=-100;
		TaperBusy:=FALSE;
		TaperDone:=FALSE;
		Error:=TRUE;
		RightTopLin_MC_Stop.Execute:=FALSE;
		RightBottomLin_MC_Stop.Execute:=FALSE;
		A_StopMC();
		fb_ton.IN:=FALSE;

END_CASE
END_IF
END_ACTION

ACTION A_TopStop:
IF TopStop THEN
TopBusy:=TRUE;
TopDone:=FALSE;
fb_ton1(PT:=t#100ms);
A_StopMC();
CASE TopState OF
	0:
		IF Top_MC_Stop.Error OR RightTopLin_MC_Stop.Error THEN
			ErrorID:=1;
			TopState:=-100;
			Top_MC_Stop.Execute:=FALSE;
			A_StopMC();
		ELSE
			TopState:=1;
		END_IF
	1:
		Top_MC_Stop.Execute:=TRUE;
		RightTopLin_MC_Stop.Execute:=TRUE;
		fb_ton1.IN:=TRUE;
		TopState:=2;
	2:
		IF  NOT Top_MC_Stop.Done OR NOT RightTopLin_MC_Stop.Done THEN
				TopState:=2;
		ELSE
			TopState:=88;
			Top_MC_Stop.Execute:=FALSE;
			RightTopLin_MC_Stop.Execute:=FALSE;
			A_StopMC();
		END_IF

	88:
		TopStop:=FALSE;
		TopState:=0;
		TopBusy:=FALSE;
		TopDone:=TRUE;
		Error:=FALSE;
		ErrorID:=0;
		fb_ton1.IN:=FALSE;

	-100:
		FB_PlcEmergencyStop();
		TopStop:=FALSE;
		TopState:=-100;
		TopBusy:=FALSE;
		TopDone:=FALSE;
		Error:=TRUE;
		Top_MC_Stop.Execute:=FALSE;
		RightTopLin_MC_Stop.Execute:=FALSE;
		A_StopMC();
		fb_ton1.IN:=FALSE;

END_CASE
END_IF
END_ACTION

END_FUNCTION_BLOCK

// ---- POUs/CommonFB/MainFB/FB_Power.TcPOU
(****************************************************************
NAME:			FB_PowerOn
DATA:			2017.2.16
VERSION:		1.0.0
DESCRIPTION:	FB_PowerOn
HISTORY:
				2017.2.16		NEW

***************************************************************)
FUNCTION_BLOCK FB_Power
VAR_INPUT
	On:BOOL;
	Off:BOOL;
	Check:BOOL;
END_VAR
VAR_OUTPUT
	FbID:DINT:=1001;
	OnState:DINT;
	OffState: INT;
	OnBusy:BOOL;
	OffBusy:BOOL;
	OnStatus:BOOL;
	OffStatus: BOOL;
	Error:BOOL;
	ErrorID:DINT;
	PowerState:BOOL;
END_VAR
VAR
	LeftTopLin_MC_Power: MC_Power;
	RightTopLin_MC_Power: MC_Power;
	LeftBottomLin_MC_Power: MC_Power;
	RightBottomLin_MC_Power: MC_Power;
	fb_ton:TON;
END_VAR

(*power on *)
IF On AND NOT Off THEN
	A_PowerOn();
(*Power Off *)
ELSIF Off AND NOT On THEN
	A_PowerOff();
END_IF
(*Check*)
IF Check THEN
	A_CheckPowerStatus();
END_IF

ACTION A_CheckPowerStatus:
A_PowerMC();
IF  LeftTopLin_MC_Power.Status AND RightTopLin_MC_Power.Status
		AND LeftBottomLin_MC_Power.Status AND RightBottomLin_MC_Power.Status THEN
	PowerState:=1;
ELSIF NOT LeftTopLin_MC_Power.Status AND NOT RightTopLin_MC_Power.Status
		AND NOT LeftBottomLin_MC_Power.Status AND NOT RightBottomLin_MC_Power.Status THEN
	PowerState:=0;
ELSE
	PowerState:=0;
	Error:=TRUE;
	ErrorID:=77;
	(*FB_PlcEmergencyStop();*)
END_IF
END_ACTION

ACTION A_PowerMC:
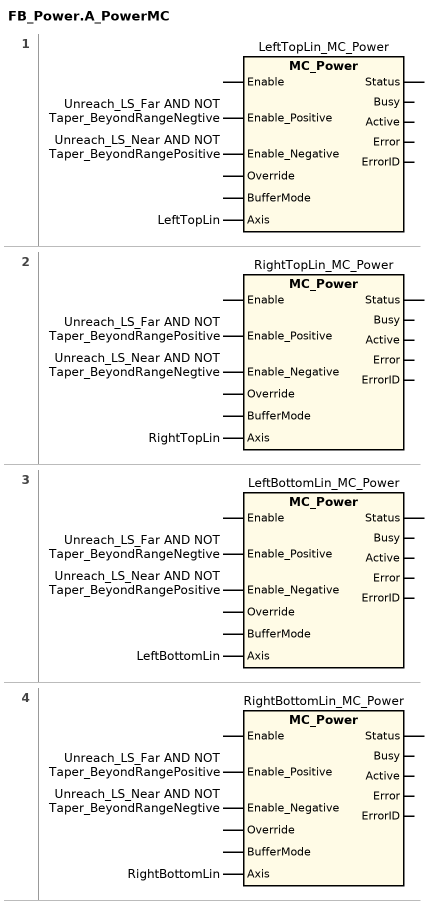
// NETWORK 1
LeftTopLin_MC_Power(
    Enable_Positive := Unreach_LS_Far AND NOT Taper_BeyondRangeNegtive,
    Enable_Negative := Unreach_LS_Near AND NOT Taper_BeyondRangePositive,
    Axis := LeftTopLin); // MC_Power

// NETWORK 2
RightTopLin_MC_Power(
    Enable_Positive := Unreach_LS_Far AND NOT Taper_BeyondRangePositive,
    Enable_Negative := Unreach_LS_Near AND NOT Taper_BeyondRangeNegtive,
    Axis := RightTopLin); // MC_Power

// NETWORK 3
LeftBottomLin_MC_Power(
    Enable_Positive := Unreach_LS_Far AND NOT Taper_BeyondRangeNegtive,
    Enable_Negative := Unreach_LS_Near AND NOT Taper_BeyondRangePositive,
    Axis := LeftBottomLin); // MC_Power

// NETWORK 4
RightBottomLin_MC_Power(
    Enable_Positive := Unreach_LS_Far AND NOT Taper_BeyondRangePositive,
    Enable_Negative := Unreach_LS_Near AND NOT Taper_BeyondRangeNegtive,
    Axis := RightBottomLin); // MC_Power
END_ACTION

ACTION A_PowerOff:
(*
IF NOT LeftTopLin_MC_Power.Status OR NOT RightTopLin_MC_Power.Status
			OR NOT LeftBottomLin_MC_Power.Status OR NOT RightBottomLin_MC_Power.Status THEN		
			LeftTopLin_MC_Power.Enable:=TRUE;
			RightTopLin_MC_Power.Enable:=TRUE;
			LeftBottomLin_MC_Power.Enable:=TRUE;
			RightBottomLin_MC_Power.Enable:=TRUE;
			A_PowerMC();
			fb_ton.IN:=TRUE;
			State:=2;
		ELSE
			ErrorID:=4;
			State:=-100;
		END_IF
*)
OffBusy:=TRUE;
CASE OffState OF
	0:
		IF NOT LeftTopLin_MC_Power.Status AND NOT RightTopLin_MC_Power.Status
			AND NOT LeftBottomLin_MC_Power.Status AND NOT RightBottomLin_MC_Power.Status THEN	
			OffState:=88;
		ELSE
			OffState:=1;
		END_IF
	1:
		LeftTopLin_MC_Power.Enable:=FALSE;
		RightTopLin_MC_Power.Enable:=FALSE;
		LeftBottomLin_MC_Power.Enable:=FALSE;
		RightBottomLin_MC_Power.Enable:=FALSE;
		A_PowerMC();
		OffState:=2;
	2:
		IF NOT LeftTopLin_MC_Power.Status AND NOT RightTopLin_MC_Power.Status
			AND NOT LeftBottomLin_MC_Power.Status AND NOT RightBottomLin_MC_Power.Status THEN	
			OffState:=88;
		ELSE
			ErrorId:=11;
			OffState:=-100;
		END_IF
	88:
		Off:=FALSE;
		OffState:=0;
		OffBusy:=FALSE;
		OnStatus:=FALSE;
		OffStatus:=TRUE;
		Error:=FALSE;
		ErrorID:=0;
	-100:
		FB_PlcEmergencyStop();
		Off:=FALSE;
		OffState:=-100;
		OffBusy:=FALSE;
		OffStatus:=FALSE;
		Error:=TRUE;

END_CASE
END_ACTION

ACTION A_PowerOn:
OnBusy:=TRUE;
fb_ton(PT:=t#0.5s);
CASE OnState OF
	0:	(*Check*)
		A_PowerMC();
		IF LeftTopLin_MC_Power.Error OR RightTopLin_MC_Power.Error
			OR LeftBottomLin_MC_Power.Error OR RightBottomLin_MC_Power.Error
			OR NOT LeftTopLin_MC_Power.Active OR NOT RightTopLin_MC_Power.Active
			OR NOT LeftBottomLin_MC_Power.Active OR NOT RightBottomLin_MC_Power.Active THEN		(*FB Error*)
			ErrorID:=1;
			OnState:=99;
		ELSIF LeftTopLin_MC_Power.Status OR RightTopLin_MC_Power.Status
			OR LeftBottomLin_MC_Power.Status OR RightBottomLin_MC_Power.Status THEN		
			ErrorID:=2;
			OnState:=-100;
		ELSIF NOT LeftTopLin_MC_Power.Status OR NOT RightTopLin_MC_Power.Status
			OR NOT LeftBottomLin_MC_Power.Status OR NOT RightBottomLin_MC_Power.Status THEN	
			OnState:=1;
		ELSE
			ErrorID:=3;
			OnState:=-100;
		END_IF
	1:	(*Execute*)
		IF NOT LeftTopLin_MC_Power.Status OR NOT RightTopLin_MC_Power.Status
			OR NOT LeftBottomLin_MC_Power.Status OR NOT RightBottomLin_MC_Power.Status THEN		
			LeftTopLin_MC_Power.Enable:=TRUE;
			RightTopLin_MC_Power.Enable:=TRUE;
			LeftBottomLin_MC_Power.Enable:=TRUE;
			RightBottomLin_MC_Power.Enable:=TRUE;
			A_PowerMC();
			fb_ton.IN:=TRUE;
			OnState:=2;
		ELSE
			ErrorID:=4;
			OnState:=-100;
		END_IF
	2:	(*Wait*)
		A_PowerMC();
		IF NOT LeftTopLin_MC_Power.Status OR NOT RightTopLin_MC_Power.Status
			OR NOT LeftBottomLin_MC_Power.Status OR NOT RightBottomLin_MC_Power.Status THEN		
			IF NOT fb_ton.Q THEN
				OnState:=2;
			ELSE
				ErrorID:=8;
				OnState:=99;
			END_IF
		ELSIF  LeftTopLin_MC_Power.Status AND RightTopLin_MC_Power.Status
			AND LeftBottomLin_MC_Power.Status AND RightBottomLin_MC_Power.Status THEN			
				OnState:=88;
		ELSE
				ErrorID:=9;
				OnState:=-100;
		END_IF
	88:
		On:=FALSE;
		OnState:=0;
		OnBusy:=FALSE;
		OnStatus:=TRUE;
		OffStatus:=FALSE;
		Error:=FALSE;
		ErrorID:=0;
		fb_ton.IN:=FALSE;
	99:
		On:=FALSE;
		OnState:=99;
		OnBusy:=FALSE;
		OnStatus:=FALSE;
		Error:=TRUE;
		LeftTopLin_MC_Power.Enable:=FALSE;
		RightTopLin_MC_Power.Enable:=FALSE;
		LeftBottomLin_MC_Power.Enable:=FALSE;
		RightBottomLin_MC_Power.Enable:=FALSE;
		fb_ton.IN:=FALSE;
	-100:
		FB_PlcEmergencyStop();
		On:=FALSE;
		OnState:=-100;
		OnBusy:=FALSE;
		OnStatus:=FALSE;
		Error:=TRUE;
		LeftTopLin_MC_Power.Enable:=FALSE;
		RightTopLin_MC_Power.Enable:=FALSE;
		LeftBottomLin_MC_Power.Enable:=FALSE;
		RightBottomLin_MC_Power.Enable:=FALSE;
		fb_ton.IN:=FALSE;

END_CASE
END_ACTION

END_FUNCTION_BLOCK

// ---- POUs/2.SingleMotorMode/TaperMode/TaperMode.TcPOU
PROGRAM TaperMode
VAR
	(*key Command*)
	TaperLargePositionNew:LREAL;
	TaperLargePositionActual: LREAL;
	TaperPositionNew:LREAL;
	TaperVelocityNew:LREAL;
	btn_TaperMove:BOOL;
	btn_TaperStop:BOOL;
	(*Var*)
	fb_ton1:TON;
	fb_ton2:TON;
	(*Status*)
	State:DINT;
	Busy:BOOL;
	InitDone:BOOL;
	Error:BOOL;
	ErrorID:DINT;
	m_state: DINT;
	s_state: DINT;
	ton_t: TON;
	range_state: DINT;
	d_state: DINT;
	(*¼ì²âµ½ÏÞÎ»£¬»Ö¸´Move×´Ì¬*)
	FTrig_ReachLS: F_TRIG;
	FTrig_btn_GapMove: F_TRIG;
END_VAR

TaperPositionActual:=((Pos_RightTopLin+Pos_RighTBottomLin)-(Pos_LeftTopLin+Pos_LeftBottomLin))/2;	
TaperVelocityActual:=(Velo_RightTopLin+Velo_RightBottomLin)/2;
TaperLargePositionActual:=TaperPositionActual+(Pos_LeftTopLin+Pos_LeftBottomLin)/2;					
TaperLargePositionNew:=TaperPositionNew+(Pos_LeftTopLin+Pos_LeftBottomLin)/2;					
(*********************************************************************Monitor All Carrirt Position***********************************************)
A_MonitoringAllAxis();
(*********************************************************************A_PosDiffDetection***********************************************)
A_PosDiffDetection();
(*********************************************************************btn_PowerOn************************************************************)
IF btn_Power AND st_Power=0 THEN
	btn_PowerOn:=TRUE;
	btn_Power:=FALSE;
END_IF
IF btn_Power AND st_Power=1 THEN
	btn_PowerOff:=TRUE;
	btn_Power:=FALSE;
END_IF
(*********************************************************************btn_PowerOn************************************************************)
IF btn_PowerOn THEN
	A_PowerOn();
END_IF
(******************************************************ÉÏµç×´Ì¬£¬´¦ÓÚñîºÏ×´Ì¬£¬ESTOP***********************************************)
IF NOT btn_PowerOff THEN
	IF st_Power=1 AND st_Couple<>0THEN
		Error:=TRUE;
		ErrorID:=101;
		FB_PlcEmergencyStop();
		LED_Error:=TRUE;
	END_IF
END_IF
(*********************************************************************btn_Move*****************************************************************)
IF InitDone THEN
	IF btn_TaperMove THEN
		CASE m_state OF
			0:
				FB_Move.Mode:=3;						
				FB_Move.CoupleState:=st_Couple;			
				FB_Move.PowerState:=st_Power;		
				FB_Move.TaperMove:=TRUE;				
				FB_Move.TaperPosition:=TaperLargePositionNew;	
				FB_Move.TaperVelocity:=TaperVelocityNew;	
				FB_Move();							
				m_state:=1;
			1:
				FB_Move();
				IF NOT FB_Move.TaperDone THEN			
					m_state:=1;
					LED_Run:=TRUE;
				ELSE									
					m_state:=88;
				END_IF

			88:
				btn_TaperMove:=FALSE;					
				m_state:=0;
				LED_Run:=FALSE;
		END_CASE
	END_IF
END_IF
(*******************************************************************btn_Stop********************************************************************)
IF btn_TaperStop THEN
	LED_Run:=FALSE;
	TaperMoveIndicator:=0;
	FB_Move.TaperReset:=TRUE;							
	FB_Move();											
	btn_TaperMove:=FALSE;								
	m_state:=0;										
	CASE s_state OF
			0:
				FB_Stop.Mode:=3;						
				FB_Stop.CoupleState:=st_Couple;			
				FB_Stop.PowerState:=st_Power;		
				FB_Stop.TaperStop:=TRUE;			
				FB_Stop();								
				s_state:=1;
			1:
				FB_Stop();
				IF NOT FB_Stop.TaperDone THEN			
					s_state:=1;
				ELSE									
					s_state:=88;
				END_IF
			88:
				btn_TaperStop:=FALSE;						
				FB_Move.TaperReset:=FALSE;					
				s_state:=0;
		END_CASE

END_IF
(****************************TaperMoveIndicator***************************)
IF TaperVelocityActual>0 THEN
	TaperMoveIndicator:=1;
ELSIF TaperVelocityActual<0 THEN
	TaperMoveIndicator:=-1;
ELSE
	TaperMoveIndicator:=0;
END_IF
(*********************************************************************btn_PowerOff************************************************************)
IF btn_PowerOff THEN
	A_PowerOff();
END_IF
(******************************************************************************************************************************)

FTrig_ReachLS(CLK:=Unreach_LS_Far AND Unreach_LS_Near);
IF FTrig_ReachLS.Q THEN
	btn_TaperStop:=TRUE;
END_IF

IF NOT Unreach_LS_Far AND TaperLargePositionNew-TaperLargePositionActual>0.0005 AND btn_TaperMove THEN
	btn_TaperStop:=TRUE;
END_IF
IF NOT Unreach_LS_Near AND TaperLargePositionNew-TaperLargePositionActual<0.0005 AND btn_TaperMove THEN
	btn_TaperStop:=TRUE;
END_IF

ACTION A_MonitoringAllAxis:
(****************************************************************
NAME:			A_MonitoringAllAxis
DATA:			2017.3.20
VERSION:		1.0.0
DESCRIPTION:	

HISTORY:
				2017.3.27		NEW

***************************************************************)
(*********************************************************************************************************************************************************************)

IF  LeftTopLin.Status.Moving OR LeftBottomLin.Status.Moving THEN
	btn_TaperStop:=TRUE;
	FB_PlcEmergencyStop();
	Error:=TRUE;
	ErrorID:=11;
	LED_Error:=TRUE;
END_IF

IF (RightTopLin.Status.Moving AND NOT RightBottomLin.Status.Moving) OR (NOT RightTopLin.Status.Moving AND RightBottomLin.Status.Moving) THEN
	btn_TaperStop:=TRUE;
	FB_PlcEmergencyStop();
	Error:=TRUE;
	ErrorID:=12;
	LED_Error:=TRUE;
END_IF
(*************************************************************************************************************************************************)
IF st_power<>0 THEN
IF (Pos_RightTopLin-Pos_leftTopLin>Range_TaperPos/2) OR (Pos_RightBottomLin-Pos_leftBottomLin>Range_TaperPos/2) THEN
	Taper_BeyondRangePositive:=TRUE;
ELSE
	Taper_BeyondRangePositive:=FALSE;
END_IF
IF  (Pos_leftTopLin-Pos_RightTopLin>Threshold_TaperTopPos) OR (Pos_leftBottomLin-Pos_RightBottomLin>Threshold_TaperBottomPos) THEN
	Taper_BeyondRangeNegtive:=TRUE;
ELSE
	Taper_BeyondRangeNegtive:=FALSE;
END_IF
IF ABS(Pos_LeftTopLin-Pos_LeftBottomLin)>Threshold_TaperLeftPos  THEN
	btn_TaperStop:=TRUE;
	FB_PlcEmergencyStop();
	Error:=TRUE;
	ErrorID:=13;
	LED_Error:=TRUE;
ELSIF  ABS(Velo_leftTopLin-Velo_LeftBottomLin)>Threshold_TaperLeftVelo THEN
	(*btn_TaperStop:=TRUE;
	FB_PlcEmergencyStop();*)
	Error:=TRUE;
	ErrorID:=14;
END_IF
IF ABS(Pos_RightTopLin-Pos_RightBottomLin)>Threshold_TaperRightPos  THEN
	btn_TaperStop:=TRUE;
	FB_PlcEmergencyStop();
	Error:=TRUE;
	ErrorID:=15;
	LED_Error:=TRUE;
ELSIF  ABS(Velo_RightTopLin-Velo_RightBottomLin)>Threshold_TaperRightVelo THEN
	(*btn_TaperStop:=TRUE;
	FB_PlcEmergencyStop();*)
	Error:=TRUE;
	ErrorID:=16;
END_IF
END_IF
(************************************************************************************************************)
END_ACTION

ACTION A_PosDiffDetection:
IF ABS(PosDiff_LeftTopLin_actual-PosDiff_RightTopLin_actual)>0.2 THEN
	ErrorID:=51;
	Error:=TRUE;
	btn_TaperStop:=TRUE;
	FB_PlcEmergencyStop();
	LED_Error:=TRUE;
ELSIF ABS(PosDiff_LeftBottomLin_actual-PosDiff_RightBottomLin_actual)>0.2 THEN
	ErrorID:=53;
	Error:=TRUE;
	btn_TaperStop:=TRUE;
	FB_PlcEmergencyStop();
	LED_Error:=TRUE;
END_IF
END_ACTION

ACTION A_PowerOff:
CASE d_state OF
		0:(*PowerOff*)
			FB_Power(Off:=TRUE);
				d_state:=1;
		1:
			IF NOT FB_power.OffStatus THEN
				d_state:=1;
			ELSE
				d_state:=88;
			END_IF
		88:(*ResetAllState*)
			btn_PowerOn:=FALSE;
			btn_TaperMove:=FALSE;
			btn_TaperStop:=FALSE;
			fb_ton1.IN:=FALSE;
			fb_ton2.IN:=FALSE;
			ton_t.IN:=FALSE;
			State:=0;
			Busy:=FALSE;
			InitDone:=FALSE;
			Error:=FALSE;
			ErrorID:=0;
			m_state:=0;
			s_state:=0;
			btn_PowerOff:=FALSE;
			d_state:=0;
			LED_Error:=FALSE;
			LED_Run:=FALSE;
END_CASE
END_ACTION

ACTION A_powerOn:
(****************************************************************
NAME:			A_SetAxisPositionAndPowerOn
DATA:			2017.3.27
VERSION:		1.0.0
DESCRIPTION:	

HISTORY:
				2017.3.27		NEW

***************************************************************)
fb_ton2(PT:=t#0.5s);
CASE State OF
	0:	(*FB_Power_On*)
		FB_Power(On:=TRUE);
		fb_ton2.IN:=TRUE;
		State:=1;
	1:	(*wait*)
		FB_power();
		IF NOT FB_power.OnStatus THEN		(*FB_Power_OnÃ»ÓÐÖ´ÐÐÍê£¬wait£¬³¬Ê±FB Error*)
			IF NOT fb_ton2.Q THEN
				State:=1;
			ELSE
				ErrorID:=1;
				State:=99;
			END_IF
		ELSE
			State:=88;
		END_IF
	88:	(*All Done*)
		btn_PowerOn:=FALSE;
		State:=0;
		Error:=FALSE;
		ErrorID:=0;
		Busy:=FALSE;
		InitDone:=TRUE;
		FB_power.On:=FALSE;
		fb_ton1.IN:=FALSE;
		fb_ton2.IN:=FALSE;
	99:
		btn_PowerOn:=FALSE;
		State:=99;
		Error:=TRUE;
		Busy:=FALSE;
		InitDone:=FALSE;
		FB_Power.On:=FALSE;
		fb_ton1.IN:=FALSE;
		fb_ton2.IN:=FALSE;
		LED_Error:=TRUE;
END_CASE
END_ACTION

END_PROGRAM

// ---- POUs/1.CarrierMode/GapMode/GapMode.TcPOU
PROGRAM GapMode
VAR
	(*GapMode*)
	GapPositionNew:LREAL:=20;
	GapVelocityNew:LREAL:=1;
	btn_GapMove:BOOL;
	btn_GapStop:BOOL;
	(*Var*)
	fb_ton1:TON;
	fb_ton2:TON;
	fb_ton3:TON;
	(*Status*)
	State:DINT;
	Busy:BOOL;
	InitDone:BOOL;
	(*FB*)

	m_state: DINT;
	s_state: DINT;
	(*¼ì²âµ½ÏÞÎ»£¬»Ö¸´Move×´Ì¬*)
	FTrig_ReachLS: F_TRIG;
	FTrig_btn_GapMove: F_TRIG;
	GapOutRange: BOOL;
	(*PowerOff*)
	d_state: DINT;
	LL: LREAL;
	LL2: LREAL;
	BB:LREAL;
	AA:LREAL;
	CC:LREAL;
	DD:LREAL;
	btn_Power: BOOL;
END_VAR

GapPositionActual:=(Pos_LeftTopLin+Pos_LeftBottomLin+Pos_RightTopLIn+Pos_RightBottomLIn)/2;
GapVelocityActual:=(Velo_LeftTopLin+Velo_LeftBottomLin+Velo_RightTopLIn+Velo_RightBottomLIn)/2;
(*********************************************************************btn_PowerOn************************************************************)
IF btn_Power AND st_Power=0 THEN
	btn_PowerOn:=TRUE;
	btn_Power:=FALSE;
END_IF
IF btn_Power AND st_Power=1 THEN
	btn_PowerOff:=TRUE;
	btn_Power:=FALSE;
END_IF
(*********************************************************************btn_PowerOn************************************************************)
IF btn_PowerOn THEN
	A_CoupleAxisAndPowerOn();
END_IF
(******************************************************ÉÏµç×´Ì¬£¬²»´¦ÓÚñîºÏ×´Ì¬£¬ESTOP***********************************************)
IF NOT btn_PowerOff THEN
	IF st_Power=1 AND st_Couple<>1THEN
		Error:=TRUE;
		ErrorID:=101;
		FB_PlcEmergencyStop();
		LED_Error:=TRUE;
	END_IF
END_IF
(*********************************************************************Monitor All Carrirt Position***********************************************)
A_MonitoringAllAxis();
(*********************************************************************A_PosDiffDetection***********************************************)
A_PosDiffDetection();
(*********************************************************************btn_Move*****************************************************************)
IF InitDone THEN
	IF btn_GapMove THEN
		CASE m_state OF
			0:
				FB_Move.Mode:=1;				
				FB_Move.CoupleState:=st_Couple;			
				FB_Move.PowerState:=st_Power;			
				FB_Move.GapMove:=TRUE;				(*Execute TRUE*)
				FB_Move.GapPosition:=GapPositionNew;	
				FB_Move.GapVelocity:=GapVelocityNew;	
				FB_Move();								
				IF GapPositionNew-GapPositionActual>0.001 THEN
					GapMoveIndicator:=1;
				ELSIF GapPositionNew-GapPositionActual<0.001 THEN
					GapMoveIndicator:=-1;
				ELSE
					GapMoveIndicator:=0;
				END_IF
				m_state:=1;
			1:
				FB_Move();
				IF NOT FB_Move.GapDone THEN		
					Led_Run:=TRUE;
					m_state:=1;

				ELSE								
					m_state:=88;
				END_IF
			88:
				btn_GapMove:=FALSE;				
				Led_Run:=FALSE;
				m_state:=0;
		END_CASE
	END_IF
END_IF
(*******************************************************************btn_Stop********************************************************************)
IF btn_GapStop THEN
	Led_Run:=FALSE;
	GapMoveIndicator:=0;
	FB_Move.GapReset:=TRUE;							
	FB_Move();										
	btn_GapMove:=FALSE;							
	m_state:=0;										
	CASE s_state OF
			0:
				FB_Stop.Mode:=1;							
				FB_Stop.CoupleState:=st_Couple;		
				FB_Stop.PowerState:=st_Power;			
				FB_Stop.GapStop:=TRUE;					
				FB_Stop();							
				s_state:=1;
			1:
				FB_Stop();
				IF NOT FB_Stop.GapDone THEN		
					s_state:=1;
				ELSE								
					s_state:=88;
				END_IF
			88:
				btn_GapStop:=FALSE;						
				FB_Move.GapReset:=FALSE;			
				s_state:=0;
		END_CASE

END_IF
(*********************************************************************btn_PowerOff************************************************************)
IF btn_PowerOff THEN
	A_DecoupleAndPowerOff();
END_IF
(***********************************************************************************************************************)

FTrig_ReachLS(CLK:=Unreach_LS_Far AND Unreach_LS_Near);
IF FTrig_ReachLS.Q THEN
	btn_GapStop:=TRUE;
END_IF
IF NOT Unreach_LS_Far AND GapPositionNew-GapPositionActual>0.0005 AND btn_GapMove THEN
	btn_GapStop:=TRUE;
END_IF
IF NOT Unreach_LS_Near AND GapPositionNew-GapPositionActual<0.0005 AND btn_GapMove THEN
	btn_GapStop:=TRUE;
END_IF

ACTION A_CoupleAxisAndPowerOn:
(****************************************************************
NAME:			A_SetAxisPositionAndCoupleAxisAndPowerOn
DATA:			2017.2.16
VERSION:		1.0.0
DESCRIPTION:	

HISTORY:
				2017.2.16		NEW

***************************************************************)
fb_ton2(PT:=t#0.5s);
fb_ton3(PT:=t#0.5s);
FB_CoupleAxis();
CASE State OF
	0:	(*FB_Couple_Axis*)
		FB_CoupleAxis(Execute:=TRUE);
		fb_ton2.IN:=TRUE;
		State:=1;
	1:	(*wait*)

		IF NOT FB_CoupleAxis.InGear THEN	
			IF NOT fb_ton1.Q THEN
				State:=1;
			ELSE
				ErrorID:=1;
				State:=99;
			END_IF
		ELSE
			State:=2;
		END_IF
	2:	(*FB_Power_On*)
		FB_CoupleAxis.Execute:=FALSE;
		FB_Power(On:=TRUE);
		fb_ton3.IN:=TRUE;
		State:=3;
	3:	(*wait*)
		FB_power();
		IF NOT FB_power.OnStatus THEN		
			IF NOT fb_ton3.Q THEN
				State:=3;
			ELSE
				ErrorID:=2;
				State:=99;
			END_IF
		ELSE
			State:=88;
		END_IF
	88:	(*All Done*)
		btn_PowerOn:=FALSE;
		State:=0;
		Error:=FALSE;
		ErrorID:=0;
		Busy:=FALSE;
		InitDone:=TRUE;

		FB_power.On:=FALSE;
		fb_ton1.IN:=FALSE;
		fb_ton2.IN:=FALSE;
		fb_ton3.IN:=FALSE;
		LED_Error:=FALSE;
	99:
		btn_PowerOn:=FALSE;
		State:=99;
		Error:=TRUE;
		Busy:=FALSE;
		InitDone:=FALSE;
		fb_ton1.IN:=FALSE;
		fb_ton2.IN:=FALSE;
		fb_ton3.IN:=FALSE;
		LED_Error:=TRUE;
END_CASE
END_ACTION

ACTION A_DecoupleAndPowerOff:
FB_DecoupleAxis();
CASE d_state OF
		0:(*Decouple*)
			FB_DecoupleAxis.Execute:=TRUE;
			FB_DecoupleAxis();
			d_state:=1;
		1:
			IF NOT FB_DecoupleAxis.OutGear THEN
				d_state:=1;
			ELSE
				d_state:=2;
			END_IF
		2:(*PowerOff*)
			FB_Power(Off:=TRUE);
				d_state:=3;
		3:
			IF NOT FB_power.OffStatus THEN
				d_state:=3;
			ELSE
				d_state:=88;
			END_IF
		88:(*ResetAllState*)
			btn_PowerOn:=FALSE;
			btn_GapMove:=FALSE;
			btn_GapStop:=FALSE;
			fb_ton1.IN:=FALSE;
			fb_ton2.IN:=FALSE;
			fb_ton3.IN:=FALSE;
			State:=0;
			Busy:=FALSE;
			InitDone:=FALSE;
			Error:=FALSE;
			ErrorID:=0;
			m_state:=0;
			s_state:=0;
			btn_PowerOff:=FALSE;
			d_state:=0;
			FB_DecoupleAxis.Execute:=FALSE;
			FB_DecoupleAxis.Reset:=TRUE;
			FB_DecoupleAxis();
			FB_CoupleAxis.Execute:=FALSE;
			FB_CoupleAxis.Reset:=TRUE;
			FB_CoupleAxis();
			Led_Run:=FALSE;
			Led_Error:=FALSE;
END_CASE
END_ACTION

ACTION A_MonitoringAllAxis:
(****************************************************************
NAME:			A_MonitoringAllAxis
DATA:			2017.2.24
VERSION:		1.0.0
DESCRIPTION:	
		
HISTORY:
				2017.2.24		NEW

***************************************************************)
(*****************************************************************************************************************************************************************)

IF  (LeftTopLin.Status.Moving AND NOT RightTopLin.Status.Moving AND NOT  LeftBottomLin.Status.Moving AND NOT RightBottomLin.Status.Moving)
	OR (NOT LeftTopLin.Status.Moving AND RightTopLin.Status.Moving AND NOT LeftBottomLin.Status.Moving AND NOT RightBottomLin.Status.Moving)
	OR (NOT LeftTopLin.Status.Moving AND NOT RightTopLin.Status.Moving AND LeftBottomLin.Status.Moving AND NOT  RightBottomLin.Status.Moving)
	OR (NOT LeftTopLin.Status.Moving AND NOT RightTopLin.Status.Moving AND NOT LeftBottomLin.Status.Moving AND RightBottomLin.Status.Moving) THEN
		btn_GapStop:=TRUE;
		FB_PlcEmergencyStop();
		Error:=TRUE;
		ErrorID:=11;
		LED_Error:=TRUE;

(*
ELSIF  (LeftTopLin.Status.Moving AND RightTopLin.Status.Moving AND NOT LeftBottomLin.Status.Moving AND NOT RightBottomLin.Status.Moving)
	OR  (LeftTopLin.Status.Moving AND NOT RightTopLin.Status.Moving AND LeftBottomLin.Status.Moving AND NOT RightBottomLin.Status.Moving)
	OR  (LeftTopLin.Status.Moving AND NOT RightTopLin.Status.Moving AND NOT LeftBottomLin.Status.Moving AND RightBottomLin.Status.Moving)
	OR  (NOT LeftTopLin.Status.Moving AND RightTopLin.Status.Moving AND LeftBottomLin.Status.Moving AND NOT RightBottomLin.Status.Moving)
	OR  (NOT LeftTopLin.Status.Moving AND RightTopLin.Status.Moving AND NOT LeftBottomLin.Status.Moving AND RightBottomLin.Status.Moving)
	OR  (NOT LeftTopLin.Status.Moving AND NOT RightTopLin.Status.Moving AND LeftBottomLin.Status.Moving AND RightBottomLin.Status.Moving) THEN
		btn_GapStop:=TRUE;
		FB_PlcEmergencyStop();
		Error:=TRUE;
		ErrorID:=12;
		LED_Error:=TRUE;
*)

ELSIF  (NOT LeftTopLin.Status.Moving AND RightTopLin.Status.Moving AND LeftBottomLin.Status.Moving AND RightBottomLin.Status.Moving)
	OR  (LeftTopLin.Status.Moving AND NOT RightTopLin.Status.Moving AND LeftBottomLin.Status.Moving AND RightBottomLin.Status.Moving)
	OR  (LeftTopLin.Status.Moving AND RightTopLin.Status.Moving AND NOT  LeftBottomLin.Status.Moving AND RightBottomLin.Status.Moving)
	OR  (LeftTopLin.Status.Moving AND RightTopLin.Status.Moving AND LeftBottomLin.Status.Moving AND NOT RightBottomLin.Status.Moving) THEN
		btn_GapStop:=TRUE;
		FB_PlcEmergencyStop();
		Error:=TRUE;
		ErrorID:=13;
		LED_Error:=TRUE;
END_IF
(*************************************************************************************2.4Öá¹âÕ¤³ßÎ»ÖÃ¡¢ËÙ¶È¶Ô±È¼ì²é**********************************************************************)
IF  st_Power<>0 THEN

		Diff_TopPos_actual:=Pos_leftTopLin-Pos_RightTopLin;
		Diff_TopVelo_actual:=Velo_leftTopLin-Velo_RightTopLin;
IF ABS(Pos_leftTopLin-Pos_RightTopLin)>Threshold_BCTopPos THEN
		btn_GapStop:=TRUE;
		FB_PlcEmergencyStop();
		Error:=TRUE;
		ErrorID:=14;
		LED_Error:=TRUE;
ELSIF ABS(Velo_leftTopLin-Velo_RightTopLin)>Threshold_BCTopVelo  THEN
		(*btn_GapStop:=TRUE;
		FB_PlcEmergencyStop();*)
		AA:=Velo_leftTopLin-Velo_RightTopLin;
		Error:=TRUE;
		ErrorID:=15;

ELSIF ABS(Pos_LeftBottomLin-Pos_RightBottomLin)>Threshold_BCBottomPos THEN
		btn_GapStop:=TRUE;
		FB_PlcEmergencyStop();
		Error:=TRUE;
		ErrorID:=16;
		LED_Error:=TRUE;
ELSIF ABS(Velo_leftBottomLin-Velo_RightBottomLin)>Threshold_BCBottomVelo  THEN
		(*btn_GapStop:=TRUE;
		FB_PlcEmergencyStop();*)
		BB:=Velo_leftBottomLin-Velo_RightBottomLin;
		Error:=TRUE;
		ErrorID:=17;

ELSIF ABS(Pos_LeftTopLin-Pos_LeftBottomLin)>Threshold_BCLeftPos  THEN
		btn_GapStop:=TRUE;
		FB_PlcEmergencyStop();
		Error:=TRUE;
		ErrorID:=18;
		LED_Error:=TRUE;
ELSIF  ABS(Velo_LeftTopLin-Velo_LeftBottomLin)>Threshold_BCLeftVelo THEN
		(*btn_GapStop:=TRUE;
		FB_PlcEmergencyStop();*)
		CC:=Velo_LeftTopLin-Velo_LeftBottomLin;
		Error:=TRUE;
		ErrorID:=19;

ELSIF ABS(Pos_RightTopLin-Pos_RightBottomLin)>Threshold_BCRightPos  THEN
		btn_GapStop:=TRUE;
		FB_PlcEmergencyStop();
		Error:=TRUE;
		ErrorID:=20;
		LED_Error:=TRUE;
ELSIF  ABS(Velo_RightTopLin-Velo_RightBottomLin)>Threshold_BCRightVelo THEN
		(*btn_GapStop:=TRUE;
		FB_PlcEmergencyStop();*)
		DD:=Velo_RightTopLin-Velo_RightBottomLin;
		Error:=TRUE;
		ErrorID:=21;
END_IF
END_IF
		LL:=Velo_LeftTopLin-Velo_LeftBottomLin;
		LL2:=Velo_RightTopLin-Velo_RightBottomLin;
(*********************************************************************************3.Ã¿Öá¹âÕ¤ºÍ±àÂëÆ÷Î»ÖÃ¶Ô±È¼ì²é**********************************************************************)
END_ACTION

ACTION A_PosDiffDetection:
IF ABS(PosDiff_LeftTopLin_actual-PosDiff_RightTopLin_actual)>0.2 THEN		(*ÉÏÖá×óÓÒÊµ¼ÊÎ»ÖÃÖ®²î*)
	ErrorID:=51;
	Error:=TRUE;
	btn_GapStop:=TRUE;
	FB_PlcEmergencyStop();
	LED_Error:=TRUE;
ELSIF ABS(PosDiff_LeftBottomLin_actual-PosDiff_RightBottomLin_actual)>0.2 THEN
	ErrorID:=53;
	Error:=TRUE;
	btn_GapStop:=TRUE;
	FB_PlcEmergencyStop();
	LED_Error:=TRUE;
END_IF
END_ACTION

END_PROGRAM

// ---- POUs/CommonFB/MainFB/FB_DecoupleAxis.TcPOU
(****************************************************************
NAME:			FB_DecoupleAxis
DATA:			2017.2.24
VERSION:		1.0.0
DESCRIPTION:	FB_DecoupleAxis
HISTORY:
				2017.2.16		NEW

***************************************************************)
FUNCTION_BLOCK FB_DecoupleAxis
VAR_INPUT
	Execute:BOOL;
	Reset:BOOL;
END_VAR
VAR_OUTPUT
	FbID:DINT:=1001;
	State:DINT;
	Busy:BOOL;
	OutGear:BOOL;
	Error:BOOL;
	ErrorID:DINT;
END_VAR
VAR
	Top_MC_GearOut: MC_GearOut;
	Bottom_MC_GearOut: MC_GearOut;
	fb_ton: TON;
END_VAR

IF Execute THEN
Busy:=TRUE;
fb_ton(PT:=t#0.1s);
CASE State OF
	0:	(*Decouple Check*)
		IF  LeftTopLin.NcToPlc.CoupleState=0 AND RightTopLin.NcToPlc.CoupleState=0
			AND LeftBottomLin.NcToPlc.CoupleState=0 AND RightBottomLin.NcToPlc.CoupleState=0 THEN	
			State:=88;
		ELSIF LeftTopLin.NcToPlc.CoupleState<>1 AND RightTopLin.NcToPlc.CoupleState<>3
			AND LeftBottomLin.NcToPlc.CoupleState<>1 AND RightBottomLin.NcToPlc.CoupleState<>3 THEN		
			ErrorID:=1;
			State:=-100;
		ELSIF Top_MC_GearOut.Error OR Bottom_MC_GearOut.Error THEN		(*FB ´íÎó*)
			ErrorID:=2;
			State:=99;
		ELSIF LeftTopLin.NcToPlc.CoupleState=1 AND RightTopLin.NcToPlc.CoupleState=3
			AND LeftBottomLin.NcToPlc.CoupleState=1 AND RightBottomLin.NcToPlc.CoupleState=3 THEN		
			State:=1;
		END_IF
	1:	(*Decouple*)
		IF LeftTopLin.NcToPlc.CoupleState=1 AND RightTopLin.NcToPlc.CoupleState=3
			AND LeftBottomLin.NcToPlc.CoupleState=1 AND RightBottomLin.NcToPlc.CoupleState=3 THEN		
			Top_MC_GearOut.Execute:=TRUE;
			Bottom_MC_GearOut.Execute:=TRUE;
			A_DecoupleMC();
			fb_ton.IN:=TRUE;
		ELSIF LeftTopLin.NcToPlc.CoupleState=0 AND RightTopLin.NcToPlc.CoupleState=0
			AND LeftBottomLin.NcToPlc.CoupleState=0 AND RightBottomLin.NcToPlc.CoupleState=0 THEN	
			State:=88;
		ELSE
			ErrorID:=3;
			State:=-100;
		END_IF
	2:	(*Decouple Wait*)
		A_DecoupleMC();
		IF NOT Top_MC_GearOut.Done OR NOT Bottom_MC_GearOut.Done THEN	
			IF NOT fb_ton.Q THEN
				State:=2;
			ELSE
				ErrorID:=4;
				State:=99;
			END_IF
		ELSIF Top_MC_GearOut.Done AND Bottom_MC_GearOut.Done
			AND LeftTopLin.NcToPlc.CoupleState=0 AND RightTopLin.NcToPlc.CoupleState=0
			AND LeftBottomLin.NcToPlc.CoupleState=0 AND RightBottomLin.NcToPlc.CoupleState=0 THEN		
			State:=88;
		ELSE
			ErrorID:=5;
			State:=-100;
		END_IF
	88:	(*Done*)
		Execute:=FALSE;
		State:=0;
		Busy:=FALSE;
		OutGear:=TRUE;
		Error:=FALSE;
		ErrorID:=0;
		Top_MC_GearOut.Execute:=FALSE;
		Bottom_MC_GearOut.Execute:=FALSE;
		A_DecoupleMC();
		fb_ton.IN:=FALSE;
	99:	(*FB Error*)
		Execute:=FALSE;
		State:=99;
		Busy:=FALSE;
		OutGear:=FALSE;
		Error:=TRUE;
		Top_MC_GearOut.Execute:=FALSE;
		Bottom_MC_GearOut.Execute:=FALSE;
		A_DecoupleMC();
		fb_ton.IN:=FALSE;
	-100:	(*EStop Error*)
		FB_PlcEmergencyStop();
		Execute:=FALSE;
		State:=-100;
		Busy:=FALSE;
		OutGear:=FALSE;
		Error:=TRUE;
		Top_MC_GearOut.Execute:=FALSE;
		Bottom_MC_GearOut.Execute:=FALSE;
		A_DecoupleMC();
		fb_ton.IN:=FALSE;

END_CASE
END_IF
IF Reset THEN
		Execute:=FALSE;
		State:=0;
		Busy:=FALSE;
		OutGear:=FALSE;
		Error:=FALSE;
		ErrorID:=0;
		Top_MC_GearOut.Execute:=FALSE;
		Bottom_MC_GearOut.Execute:=FALSE;
		A_DecoupleMC();
		fb_ton.IN:=FALSE;
		Reset:=FALSE;
END_IF

ACTION A_DecoupleMC:
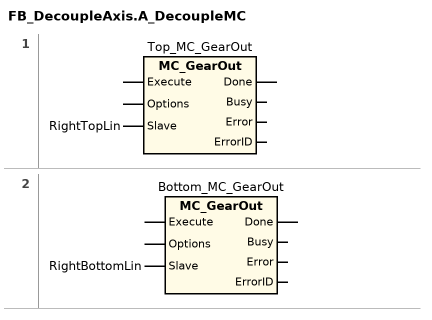
// NETWORK 1
Top_MC_GearOut(Slave := RightTopLin); // MC_GearOut

// NETWORK 2
Bottom_MC_GearOut(Slave := RightBottomLin); // MC_GearOut
END_ACTION

END_FUNCTION_BLOCK

// ---- POUs/2.SingleMotorMode/DebugMode/DebugMode.TcPOU
PROGRAM DebugMode
VAR
(* Common*)
	d_state: DINT;(*PowerOffState*)
	InitDone:BOOL;
	Busy: BOOL;
	fb_ton: TON;
	PowerState: INT;(*PowerOnState*)
	ton_t: TON;
(*Key Command*)
	LeftTopLinPositionNew:LREAL;
	LeftTopLinVelocityNew:LREAL:=0.02;
	btn_LeftTopLinMove:BOOL;
	btn_LeftTopLinStop:BOOL;
	RightTopLinPositionNew:LREAL;
	RightTopLinVelocityNew:LREAL:=0.02;
	btn_RightTopLinMove:BOOL;
	btn_RightTopLinStop:BOOL;
	LeftBottomLinPositionNew:LREAL;
	LeftBottomLinVelocityNew:LREAL:=0.02;
	btn_LeftBottomLinMove:BOOL;
	btn_LeftBottomLinStop:BOOL;
	RightBottomLinPositionNew:LREAL;
	RightBottomLinVelocityNew:LREAL:=0.02;
	btn_RightBottomLinMove:BOOL;
	btn_RightBottomLinStop:BOOL;
(*LeftTopLin*)
	fb_ton1_1:TON;
	fb_ton1_2:TON;
	LeftTopLinState:DINT;
	LeftTopLinBusy:BOOL;
	LeftTopLin_m_state: DINT;
	LeftTopLin_s_state: DINT;
(*RightTopLin*)
	fb_ton2_1:TON;
	fb_ton2_2:TON;
	RightTopLinState:DINT;
	RightTopLinBusy:BOOL;
	RightTopLin_m_state: DINT;
	RightTopLin_s_state: DINT;
(*LeftBottomLin*)
	fb_ton3_1:TON;
	fb_ton3_2:TON;
	LeftBottomLinState:DINT;
	LeftBottomLinBusy:BOOL;
	LeftBottomLin_m_state: DINT;
	LeftBottomLin_s_state: DINT;
(*RightBottomLin*)
	fb_ton4_1:TON;
	fb_ton4_2:TON;
	RightBottomLinState:DINT;
	RightBottomLinBusy:BOOL;
	RightBottomLin_m_state: DINT;
	RightBottomLin_s_state: DINT;


	btn_LeftTopStop: BOOL;
	(*¼ì²âµ½ÏÞÎ»£¬»Ö¸´Move×´Ì¬*)
	FTrig_ReachLS: F_TRIG;
	FTrig_btn_GapMove: F_TRIG;
	
	RTrig_LeftTopMove:R_TRIG;
	RTrig_RightTopMove:R_TRIG;
	RTrig_LeftBottomMove:R_TRIG;
	RTrig_RightBottomMove:R_TRIG;
	
END_VAR

(*********************************************************************Monitor All Carrirt Position***********************************************)
A_MonitoringAllAxis();
(*********************************************************************A_PosDiffDetection***********************************************)
A_PosDiffDetection();
//
IF st_Power=1 THEN
	InitDone:=TRUE;
END_IF
(*********************************************************************btn_PowerOn************************************************************)
IF btn_Power AND st_Power=0 THEN
	btn_PowerOn:=TRUE;
	btn_Power:=FALSE;
END_IF
IF btn_Power AND st_Power=1 THEN
	btn_PowerOff:=TRUE;
	btn_Power:=FALSE;
END_IF
(*********************************************************************btn_PowerOn************************************************************)
IF btn_PowerOn THEN
	A_PowerOn();
END_IF
(****************************************************ESTOP***********************************************)
IF NOT btn_PowerOff THEN
	IF st_Power=1 AND st_Couple<>0THEN
		Error:=TRUE;
		ErrorID:=101;
		FB_PlcEmergencyStop();
		LED_Error:=TRUE;
	END_IF
END_IF

(*********************************************************************btn_PowerOff************************************************************)
IF btn_PowerOff THEN
	A_PowerOff();
END_IF

A_Motion();
A_CheckTargetPos();


(****************************MoveIndicator***************************)
IF Velo_LeftTopLin>0 THEN
	LeftTopLinMoveIndicator:=1;
ELSIF Velo_LeftTopLin<0 THEN
	LeftTopLinMoveIndicator:=-1;
ELSE
	LeftTopLinMoveIndicator:=0;
END_IF
IF Velo_RightTopLin>0 THEN
	RightTopLinMoveIndicator:=1;
ELSIF Velo_RightTopLin<0 THEN
	RightTopLinMoveIndicator:=-1;
ELSE
	RightTopLinMoveIndicator:=0;
END_IF
IF Velo_LeftBottomLin>0 THEN
	LeftBottomLinMoveIndicator:=1;
ELSIF Velo_LeftBottomLin<0 THEN
	LeftBottomLinMoveIndicator:=-1;
ELSE
	LeftBottomLinMoveIndicator:=0;
END_IF
IF Velo_RightBottomLin>0 THEN
	RightBottomLinMoveIndicator:=1;
ELSIF Velo_RightBottomLin<0 THEN
	RightBottomLinMoveIndicator:=-1;
ELSE
	RightBottomLinMoveIndicator:=0;
END_IF
(*********************************************************************ÏÞÎ»Åö´¥×´Ì¬»Ö¸´************************************************************)
(*Èç¹û¼ì²âµ½ÏØÏÞÎ»¿ª¹ØÏÂ½µÑØ£¬»Ö¸´Move×´Ì¬*)
FTrig_ReachLS(CLK:=Unreach_LS_Far AND Unreach_LS_Near);
IF FTrig_ReachLS.Q THEN
	btn_LeftTopLinStop:=TRUE;
	btn_RightTopLinStop:=TRUE;
	btn_LeftBottomLinStop:=TRUE;
	btn_RightBottomLinStop:=TRUE;
END_IF
IF btn_LeftTopLinStop THEN
	btn_RightTopLinStop:=TRUE;
END_IF
IF btn_RightTopLinStop THEN
	btn_LeftBottomLinStop:=TRUE;
END_IF
IF btn_LeftBottomLinStop THEN
	btn_RightBottomLinStop:=TRUE;
END_IF

IF NOT Unreach_LS_Far AND LeftTopLinPositionNew-Pos_LeftTopLin>0.0005 AND btn_LeftTopLinMove THEN
	btn_LeftTopLinStop:=TRUE;
END_IF
IF NOT Unreach_LS_Near AND RightTopLinPositionNew-Pos_RightTopLin<0.0005 AND btn_RightTopLinMove THEN
	btn_RightTopLinStop:=TRUE;
END_IF
IF NOT Unreach_LS_Far AND LeftBottomLinPositionNew-Pos_LeftBottomLin>0.0005 AND btn_LeftBottomLinMove THEN
	btn_LeftBottomLinStop:=TRUE;
END_IF
IF NOT Unreach_LS_Near AND RightBottomLinPositionNew-Pos_RightBottomLin<0.0005 AND btn_RightBottomLinMove THEN
	btn_RightBottomLinStop:=TRUE;
END_IF

ACTION A_CheckTargetPos:
RTrig_LeftTopMove(CLK:=btn_LeftTopLinMove);
IF RTrig_LeftTopMove.Q THEN
	IF NOT st_Power THEN
			ErrorID:=1501;
			Error:=TRUE;
			ErrorDescription:='Plz PowerOn Frist';
			LED_Error:=TRUE;
			//RETURN;
		ELSIF ABS(LeftTopLinPositionNew-Pos_LeftTopLin)>Threshold_LeftTopPos_Debug THEN
			btn_LeftTopLinStop:=TRUE;
			btn_LeftTopLinMove:=FALSE;
			ErrorID:=1502;
			Error:=TRUE;
			ErrorDescription:='targetPos Out of range!';
			LED_Error:=TRUE;
			//RETURN;
		ELSE
			ErrorID:=0;
			Error:=FALSE;
			ErrorDescription:='';
			LED_Error:=FALSE;
		END_IF
END_IF
RTrig_RightTopMove(CLK:=btn_RightTopLinMove);
IF RTrig_RightTopMove.Q THEN
	IF NOT st_Power THEN
			ErrorID:=1503;
			Error:=TRUE;
			ErrorDescription:='Plz PowerOn Frist';
			LED_Error:=TRUE;
			//RETURN;
		ELSIF ABS(RightTopLinPositionNew-Pos_RightTopLin)>Threshold_RightTopPos_Debug THEN
			btn_RightTopLinStop:=TRUE;
			btn_RightTopLinMove:=FALSE;
			ErrorID:=1504;
			Error:=TRUE;
			ErrorDescription:='targetPos Out of range!';
			LED_Error:=TRUE;
			//RETURN;
		ELSE
			ErrorID:=0;
			Error:=FALSE;
			ErrorDescription:='';
			LED_Error:=FALSE;
		END_IF
END_IF
RTrig_LeftBottomMove(CLK:=btn_LeftBottomLinMove);
IF RTrig_LeftBottomMove.Q THEN
	IF NOT st_Power THEN
			ErrorID:=1505;
			Error:=TRUE;
			ErrorDescription:='Plz PowerOn Frist';
			LED_Error:=TRUE;
			//RETURN;
		ELSIF ABS(LeftBottomLinPositionNew-Pos_LeftBottomLin)>Threshold_LeftBottomPos_Debug THEN
			btn_LeftBottomLinStop:=TRUE;
			btn_LeftBottomLinMove:=FALSE;
			ErrorID:=1506;
			Error:=TRUE;
			ErrorDescription:='targetPos Out of range!';
			LED_Error:=TRUE;
			//RETURN;
		ELSE
			ErrorID:=0;
			Error:=FALSE;
			ErrorDescription:='';
			LED_Error:=FALSE;
		END_IF
END_IF
RTrig_RightBottomMove(CLK:=btn_RightBottomLinMove);
IF RTrig_RightBottomMove.Q THEN
	IF NOT st_Power THEN
			ErrorID:=1507;
			Error:=TRUE;
			ErrorDescription:='Plz PowerOn Frist';
			LED_Error:=TRUE;
			//RETURN;
		ELSIF ABS(RightBottomLinPositionNew-Pos_RightBottomLin)>Threshold_RightBottomPos_Debug THEN
			btn_RightBottomLinStop:=TRUE;
			btn_RightBottomLinMove:=FALSE;
			ErrorID:=1508;
			Error:=TRUE;
			ErrorDescription:='targetPos Out of range!';
			LED_Error:=TRUE;
			//RETURN;
		ELSE
			ErrorID:=0;
			Error:=FALSE;
			ErrorDescription:='';
			LED_Error:=FALSE;
		END_IF
END_IF
END_ACTION

ACTION A_monitoringAllAxis:
(****************************************************************
NAME:			A_MonitoringAllAxis
DATA:			2017.5.8
VERSION:		1.0.0
DESCRIPTION:	

HISTORY:
				2017.5.8	NEW

***************************************************************)

(******************************************************************************************************************************************************)
IF st_power<>0 THEN

IF ABS(Pos_LeftTopLin-Pos_LeftBottomLin)>Threshold_LeftPos_Debug  THEN
		btn_LeftTopLinStop:=TRUE;
		btn_RightTopLinStop:=TRUE;
		btn_LeftBottomLinStop:=TRUE;
		btn_RightBottomLInStop:=TRUE;
		FB_PlcEmergencyStop();
		Error:=TRUE;
		ErrorID:=11;
		LED_Error:=TRUE;
END_IF

IF ABS(Pos_RightTopLin-Pos_RightBottomLin)>Threshold_RightPos_Debug  THEN
		btn_LeftTopLinStop:=TRUE;
		btn_RightTopLinStop:=TRUE;
		btn_LeftBottomLinStop:=TRUE;
		btn_RightBottomLInStop:=TRUE;
		FB_PlcEmergencyStop();
		Error:=TRUE;
		ErrorID:=12;
		LED_Error:=TRUE;
END_IF

IF ABS(Pos_LeftTopLin-Pos_RightTopLin)>Threshold_TopPos_Debug  THEN
		btn_LeftTopLinStop:=TRUE;
		btn_RightTopLinStop:=TRUE;
		btn_LeftBottomLinStop:=TRUE;
		btn_RightBottomLInStop:=TRUE;
		FB_PlcEmergencyStop();
		Error:=TRUE;
		ErrorID:=13;
		LED_Error:=TRUE;
END_IF

IF ABS(Pos_LeftBottomLin-Pos_RightBottomLin)>Threshold_BottomPos_Debug  THEN
		btn_LeftTopLinStop:=TRUE;
		btn_RightTopLinStop:=TRUE;
		btn_LeftBottomLinStop:=TRUE;
		btn_RightBottomLInStop:=TRUE;
		FB_PlcEmergencyStop();
		Error:=TRUE;
		ErrorID:=14;
		LED_Error:=TRUE;
END_IF
END_IF
(*********************************************************************************3.Ã¿Öá¹âÕ¤ºÍ±àÂëÆ÷Î»ÖÃ¶Ô±È¼ì²é**********************************************************************)
END_ACTION

ACTION A_Motion:
(*********************************************************************LeftTop_MOVE*****************************************************************)
//IF InitDone THEN
	IF btn_LeftTopLinMove THEN
		CASE LeftTopLin_m_state OF
			0:
				FB_Move.Mode:=4;					
				FB_Move.CoupleState:=st_Couple;
				FB_Move.PowerState:=st_Power;		
				FB_Move.LeftTopMove:=TRUE;			
				FB_Move.LeftTopPosition:=LeftTopLinPositionNew;
				FB_Move.LeftTopVelocity:=LeftTopLinVelocityNew;	
				FB_Move();								
				LeftTopLin_m_state:=1;
			1:
				FB_Move();
				IF NOT FB_Move.LeftTopDone THEN		
					LeftTopLin_m_state:=1;
					LED_Run:=TRUE;
				ELSE							
					LeftTopLin_m_state:=88;
				END_IF

			88:
				btn_LeftTopLinMove:=FALSE;				
				LeftTopLin_m_state:=0;
				LED_Run:=FALSE;
		END_CASE
	END_IF
//END_IF
(*******************************************************************LeftTop_STOP********************************************************************)
IF btn_LeftTopLinStop OR btn_reset THEN
	LED_Run:=FALSE;
	FB_Move.LeftTopReset:=TRUE;							
	FB_Move();										
	btn_LeftTopLinMove:=FALSE;						
	LeftTopLin_m_state:=0;										
	CASE LeftTopLin_s_state OF
			0:
				FB_Stop.Mode:=4;							
				FB_Stop.CoupleState:=st_Couple;			
				FB_Stop.PowerState:=st_Power;				
				FB_Stop.LeftTopStop:=TRUE;				
				FB_Stop();							
				LeftTopLin_s_state:=1;
			1:
				FB_Stop();
				IF NOT FB_Stop.LeftTopDone THEN		
					LeftTopLin_s_state:=1;
				ELSE								
					LeftTopLin_s_state:=88;
				END_IF
			88:
				btn_LeftTopLinStop:=FALSE;					
				FB_Move.LeftTopReset:=FALSE;				
				LeftTopLin_s_state:=0;
				btn_reset:=FALSE;
		END_CASE

END_IF
(*********************************************************************RightTop_MOVE*****************************************************************)
//IF InitDone THEN
	IF btn_RightTopLinMove THEN
		CASE RightTopLin_m_state OF
			0:
				FB_Move.Mode:=4;						
				FB_Move.CoupleState:=st_Couple;			
				FB_Move.PowerState:=st_Power;			
				FB_Move.RightTopMove:=TRUE;			
				FB_Move.RightTopPosition:=RightTopLinPositionNew;	
				FB_Move.RightTopVelocity:=RightTopLinVelocityNew;	
				FB_Move();								
				RightTopLin_m_state:=1;
			1:
				FB_Move();
				IF NOT FB_Move.RightTopDone THEN		
					RightTopLin_m_state:=1;
					LED_Run:=TRUE;
				ELSE								
					RightTopLin_m_state:=88;
				END_IF

